	            IF ("gtyp_VGR".horizontal_Axis.di_Actual_Position <= ("gtyp_VGR".di_Pos_MPO_horizontal + "gtyp_VGR".horizontal_Axis.Config.di_Pos_Window))
	                AND ("gtyp_VGR".horizontal_Axis.di_Actual_Position >= ("gtyp_VGR".di_Pos_MPO_horizontal - "gtyp_VGR".horizontal_Axis.Config.di_Pos_Window))
	                AND "gtyp_VGR".horizontal_Axis.x_Position_Reached
	                AND ("gtyp_VGR".vertical_Axis.di_Actual_Position <= ("gtyp_VGR".di_Pos_MPO_vertical - "gtyp_VGR".di_Offset_Pos_MPO_vertical + "gtyp_VGR".vertical_Axis.Config.di_Pos_Window))
	                AND ("gtyp_VGR".vertical_Axis.di_Actual_Position >= ("gtyp_VGR".di_Pos_MPO_vertical - "gtyp_VGR".di_Offset_Pos_MPO_vertical - "gtyp_VGR".vertical_Axis.Config.di_Pos_Window))
	                AND "gtyp_VGR".vertical_Axis.x_Position_Reached THEN
	                "gtyp_VGR".horizontal_Axis.x_Start_Positioning := FALSE;
	                "gtyp_VGR".vertical_Axis.x_Start_Positioning := FALSE;
	                "gtyp_VGR".vertical_Axis.i_PWM := 800;
	                #li_StepCase := 520;
	            END_IF;

	        520: // MPO ready to discard - Position vertical MPO

	            IF "gtyp_MPO".x_Discard_Ready THEN
	                "gtyp_VGR".vertical_Axis.di_Target_Position := "gtyp_VGR".di_Pos_MPO_vertical;
	                "gtyp_VGR".vertical_Axis.x_Start_Positioning := TRUE;
	                "gtyp_VGR".vertical_Axis.i_PWM := 500;

	                IF ("gtyp_VGR".vertical_Axis.di_Actual_Position <= ("gtyp_VGR".di_Pos_MPO_vertical + "gtyp_VGR".vertical_Axis.Config.di_Pos_Window))
	                    AND ("gtyp_VGR".vertical_Axis.di_Actual_Position >= ("gtyp_VGR".di_Pos_MPO_vertical - "gtyp_VGR".vertical_Axis.Config.di_Pos_Window))
	                    AND "gtyp_VGR".vertical_Axis.x_Position_Reached THEN
	                    "gtyp_VGR".vertical_Axis.x_Start_Positioning := FALSE;
	                    "gtyp_VGR".vertical_Axis.i_PWM := 800;
	                    #li_StepCase := 530;
	                    "gtyp_VGR".x_MPO_Req_Discard := FALSE;
	                END_IF;
	            END_IF;

	        530: // turn off vacuum
	            "QX_VGR_ValveVacuum_Q8" := FALSE;
	            #li_StepCase := 540;

	        540: // turn off compressor
	            "QX_VGR_Compressor_Q7" := FALSE;
	            "gtyp_VGR".x_MPO_Discards := TRUE;
	            // Order State
	            "gtyp_VGR".x_Ready_For_Outsource := FALSE;
	            "gtyp_VGR".x_State_Process := TRUE;
	            "gtyp_Interface_Dashboard".Subscribe.State_Order.ldt_ts := DT_TO_LDT(#ldt_MQTT);
	            "gtyp_Interface_Dashboard".Subscribe.State_Order.s_state := 'IN_PROCESS';
	            "gtyp_Interface_Dashboard".Subscribe.State_Order.s_type := "gtyp_VGR".Workpiece.s_type;
	            #li_StepCase := 550;

	        550: // Workpiece discard accepted - Position pre vertical MPO

	            IF "gtyp_MPO".x_MPO_Discards_Accepted THEN
	                "gtyp_VGR".vertical_Axis.di_Target_Position := "gtyp_VGR".di_Pos_MPO_vertical - "gtyp_VGR".di_Offset_Pos_MPO_vertical;
	                "gtyp_VGR".vertical_Axis.x_Start_Positioning := TRUE;
	                "gtyp_VGR".vertical_Axis.i_PWM := 500;

	                IF ("gtyp_VGR".vertical_Axis.di_Actual_Position <= ("gtyp_VGR".di_Pos_MPO_vertical - "gtyp_VGR".di_Offset_Pos_MPO_vertical + "gtyp_VGR".vertical_Axis.Config.di_Pos_Window))
	                    AND ("gtyp_VGR".vertical_Axis.di_Actual_Position >= ("gtyp_VGR".di_Pos_MPO_vertical - "gtyp_VGR".di_Offset_Pos_MPO_vertical - "gtyp_VGR".vertical_Axis.Config.di_Pos_Window))
	                    AND "gtyp_VGR".vertical_Axis.x_Position_Reached THEN
	                    "gtyp_VGR".vertical_Axis.x_Start_Positioning := FALSE;
	                    "gtyp_VGR".x_MPO_Discards := FALSE;
	                    "gtyp_VGR".vertical_Axis.i_PWM := 800;
	                    #li_StepCase := 560;
	                END_IF;
	            END_IF;

	        560: // homing horizontal axis
	            "gtyp_VGR".horizontal_Axis.x_Reference := TRUE;

	            IF NOT "gtyp_VGR".horizontal_Axis.x_Referenced THEN
	                #li_StepCase := 570;
	            END_IF;

	        570: // homed horizontal axis
	            IF "gtyp_VGR".horizontal_Axis.x_Referenced THEN
	                "gtyp_VGR".horizontal_Axis.x_Reference := FALSE;
	                "gtyp_VGR".x_MPO_Discards := FALSE;
	                #li_StepCase := 580;
	            END_IF;

	        580: // wait sequence
	            #lx_Start_TON_Wait := TRUE;
	            #lt_TON_Wait := T#500ms;

	            IF #lfb_TON_Wait.Q THEN
	                "gtyp_VGR".Workpiece.s_id := '0';
	                "gtyp_VGR".Workpiece.s_state := '';
	                "gtyp_VGR".Workpiece.s_type := '';
	                FOR #li_Counter := 1 TO 8 DO
	                    "gtyp_VGR".History[#li_Counter].i_code := 0;
	                    "gtyp_VGR".History[#li_Counter].ldt_ts := DT#1990-01-01-00:00:00;
	                END_FOR;
	                #lx_Start_TON_Wait := FALSE;
	                #li_StepCase := 0;
	            END_IF;

	            (*******************************************************************************************)
	            (**************************      Procedure - store raw parts      **************************)
	            (*******************************************************************************************)

	        600:// approach pick-up position dsi with vertical, horizontal, rotate axis
	            "gtyp_VGR".horizontal_Axis.di_Target_Position := "gtyp_VGR".di_Pos_DSI_horizontal;
	            "gtyp_VGR".horizontal_Axis.x_Start_Positioning := TRUE;
	            "gtyp_VGR".vertical_Axis.di_Target_Position := "gtyp_VGR".di_Pos_DSI_Collect_vertical;
	            "gtyp_VGR".vertical_Axis.x_Start_Positioning := TRUE;
	            "gtyp_VGR".vertical_Axis.i_PWM := 500;
	            "gtyp_VGR".rotate_Axis.di_Target_Position := "gtyp_VGR".di_Pos_DSI_rotate;
	            "gtyp_VGR".rotate_Axis.x_Start_Positioning := TRUE;

	            IF ("gtyp_VGR".horizontal_Axis.di_Actual_Position <= ("gtyp_VGR".di_Pos_DSI_horizontal + "gtyp_VGR".horizontal_Axis.Config.di_Pos_Window))
	                AND ("gtyp_VGR".horizontal_Axis.di_Actual_Position >= ("gtyp_VGR".di_Pos_DSI_horizontal - "gtyp_VGR".horizontal_Axis.Config.di_Pos_Window))
	                AND "gtyp_VGR".horizontal_Axis.x_Position_Reached THEN
	                "gtyp_VGR".horizontal_Axis.x_Start_Positioning := FALSE;
	            END_IF;

	            IF ("gtyp_VGR".vertical_Axis.di_Actual_Position <= ("gtyp_VGR".di_Pos_DSI_Collect_vertical + "gtyp_VGR".vertical_Axis.Config.di_Pos_Window))
	                AND ("gtyp_VGR".vertical_Axis.di_Actual_Position >= ("gtyp_VGR".di_Pos_DSI_Collect_vertical - "gtyp_VGR".vertical_Axis.Config.di_Pos_Window))
	                AND "gtyp_VGR".vertical_Axis.x_Position_Reached THEN
	                "gtyp_VGR".vertical_Axis.x_Start_Positioning := FALSE;
	            END_IF;

	            IF ("gtyp_VGR".rotate_Axis.di_Actual_Position <= ("gtyp_VGR".di_Pos_DSI_rotate + "gtyp_VGR".rotate_Axis.Config.di_Pos_Window))
	                AND ("gtyp_VGR".rotate_Axis.di_Actual_Position >= ("gtyp_VGR".di_Pos_DSI_rotate - "gtyp_VGR".rotate_Axis.Config.di_Pos_Window))
	                AND "gtyp_VGR".rotate_Axis.x_Position_Reached THEN
	                "gtyp_VGR".rotate_Axis.x_Start_Positioning := FALSE;
	            END_IF;

	            IF ("gtyp_VGR".horizontal_Axis.di_Actual_Position <= ("gtyp_VGR".di_Pos_DSI_horizontal + "gtyp_VGR".horizontal_Axis.Config.di_Pos_Window))
	                AND ("gtyp_VGR".horizontal_Axis.di_Actual_Position >= ("gtyp_VGR".di_Pos_DSI_horizontal - "gtyp_VGR".horizontal_Axis.Config.di_Pos_Window))
	                AND "gtyp_VGR".horizontal_Axis.x_Position_Reached
	                AND ("gtyp_VGR".vertical_Axis.di_Actual_Position <= ("gtyp_VGR".di_Pos_DSI_Collect_vertical + "gtyp_VGR".vertical_Axis.Config.di_Pos_Window))
	                AND ("gtyp_VGR".vertical_Axis.di_Actual_Position >= ("gtyp_VGR".di_Pos_DSI_Collect_vertical - "gtyp_VGR".vertical_Axis.Config.di_Pos_Window))
	                AND "gtyp_VGR".vertical_Axis.x_Position_Reached
	                AND ("gtyp_VGR".rotate_Axis.di_Actual_Position <= ("gtyp_VGR".di_Pos_DSI_rotate + "gtyp_VGR".rotate_Axis.Config.di_Pos_Window))
	                AND ("gtyp_VGR".rotate_Axis.di_Actual_Position >= ("gtyp_VGR".di_Pos_DSI_rotate - "gtyp_VGR".rotate_Axis.Config.di_Pos_Window))
	                AND "gtyp_VGR".rotate_Axis.x_Position_Reached THEN
	                "gtyp_VGR".horizontal_Axis.x_Start_Positioning := FALSE;
	                "gtyp_VGR".vertical_Axis.x_Start_Positioning := FALSE;
	                "gtyp_VGR".rotate_Axis.x_Start_Positioning := FALSE;
	                "gtyp_VGR".vertical_Axis.i_PWM := 800;
	                #li_StepCase := 610;
	            END_IF;

	        610:// set status 100 raw goods delivered
	            #li_Return_LDT := RD_SYS_T(#ldt_MQTT);
	            "gtyp_VGR".Workpiece.s_state := 'RAW';
	            "gtyp_VGR".History[1].ldt_ts := DT_TO_LDT(#ldt_MQTT);
	            "gtyp_VGR".History[1].i_code := 100;
	            #li_StepCase := 620;

	        620:// wait sequence
	            #lx_Start_TON_Wait := TRUE;
	            #lt_TON_Wait := T#500ms;

	            IF #lfb_TON_Wait.Q THEN
	                #lx_Start_TON_Wait := FALSE;
	                #li_StepCase := 630;
	            END_IF;

	        630:// turn on compressor and wait
	            "QX_VGR_Compressor_Q7" := TRUE;

	            #lx_Start_TON_Wait := TRUE;
	            #lt_TON_Wait := T#500ms;

	            IF #lfb_TON_Wait.Q THEN
	                #lx_Start_TON_Wait := FALSE;
	                #li_StepCase := 640;
	            END_IF;

	        640:// turn on vacuum
	            "QX_VGR_ValveVacuum_Q8" := true;

	            #li_StepCase := 650;

	        650:// Position vertical NFC
	            #lx_State_activ := TRUE;
	            #ls_Target := 'hbw';

	            "gtyp_VGR".vertical_Axis.di_Target_Position := "gtyp_VGR".di_Pos_NFC_vertical - "gtyp_VGR".di_Offset_Pos_DSI_NFC_vertical;
	            "gtyp_VGR".vertical_Axis.x_Start_Positioning := TRUE;
	            "gtyp_VGR".vertical_Axis.i_PWM := 800;

	            IF ("gtyp_VGR".vertical_Axis.di_Actual_Position <= ("gtyp_VGR".di_Pos_NFC_vertical - "gtyp_VGR".di_Offset_Pos_DSI_NFC_vertical + "gtyp_VGR".vertical_Axis.Config.di_Pos_Window))
	                AND ("gtyp_VGR".vertical_Axis.di_Actual_Position >= ("gtyp_VGR".di_Pos_NFC_vertical - "gtyp_VGR".di_Offset_Pos_DSI_NFC_vertical - "gtyp_VGR".vertical_Axis.Config.di_Pos_Window))
	                AND "gtyp_VGR".vertical_Axis.x_Position_Reached THEN
	                "gtyp_VGR".vertical_Axis.x_Start_Positioning := FALSE;
	                #li_StepCase := 660;
	            END_IF;

	        660: // wait sequence
	            #lx_Start_TON_Wait := TRUE;
	            #lt_TON_Wait := T#500ms;

	            IF #lfb_TON_Wait.Q THEN
	                #lx_Start_TON_Wait := FALSE;
	                #li_StepCase := 670;
	            END_IF;

	        670: // Position horizontal/rotate NFC

	            "gtyp_VGR".horizontal_Axis.di_Target_Position := "gtyp_VGR".di_Pos_NFC_horizontal;
	            "gtyp_VGR".horizontal_Axis.x_Start_Positioning := TRUE;
	            "gtyp_VGR".rotate_Axis.di_Target_Position := "gtyp_VGR".di_Pos_NFC_rotate;
	            "gtyp_VGR".rotate_Axis.x_Start_Positioning := TRUE;

	            IF ("gtyp_VGR".horizontal_Axis.di_Actual_Position <= ("gtyp_VGR".di_Pos_NFC_horizontal + "gtyp_VGR".horizontal_Axis.Config.di_Pos_Window))
	                AND ("gtyp_VGR".horizontal_Axis.di_Actual_Position >= ("gtyp_VGR".di_Pos_NFC_horizontal - "gtyp_VGR".horizontal_Axis.Config.di_Pos_Window))
	                AND "gtyp_VGR".horizontal_Axis.x_Position_Reached THEN
	                "gtyp_VGR".horizontal_Axis.x_Start_Positioning := FALSE;
	            END_IF;

	            IF ("gtyp_VGR".rotate_Axis.di_Actual_Position <= ("gtyp_VGR".di_Pos_NFC_rotate + "gtyp_VGR".rotate_Axis.Config.di_Pos_Window))
	                AND ("gtyp_VGR".rotate_Axis.di_Actual_Position >= ("gtyp_VGR".di_Pos_NFC_rotate - "gtyp_VGR".rotate_Axis.Config.di_Pos_Window))
	                AND "gtyp_VGR".rotate_Axis.x_Position_Reached THEN
	                "gtyp_VGR".rotate_Axis.x_Start_Positioning := FALSE;
	            END_IF;

	            IF ("gtyp_VGR".horizontal_Axis.di_Actual_Position <= ("gtyp_VGR".di_Pos_NFC_horizontal + "gtyp_VGR".horizontal_Axis.Config.di_Pos_Window))
	                AND ("gtyp_VGR".horizontal_Axis.di_Actual_Position >= ("gtyp_VGR".di_Pos_NFC_horizontal - "gtyp_VGR".horizontal_Axis.Config.di_Pos_Window))
	                AND "gtyp_VGR".horizontal_Axis.x_Position_Reached
	                AND ("gtyp_VGR".rotate_Axis.di_Actual_Position <= ("gtyp_VGR".di_Pos_NFC_rotate + "gtyp_VGR".rotate_Axis.Config.di_Pos_Window))
	                AND ("gtyp_VGR".rotate_Axis.di_Actual_Position >= ("gtyp_VGR".di_Pos_NFC_rotate - "gtyp_VGR".rotate_Axis.Config.di_Pos_Window))
	                AND "gtyp_VGR".rotate_Axis.x_Position_Reached THEN
	                "gtyp_VGR".horizontal_Axis.x_Start_Positioning := FALSE;
	                "gtyp_VGR".rotate_Axis.x_Start_Positioning := FALSE;
	                #li_StepCase := 680;
	            END_IF;

	        680: // wait sequence
	            #lx_Start_TON_Wait := TRUE;
	            #lt_TON_Wait := T#500ms;

	            IF #lfb_TON_Wait.Q THEN
	                #lx_Start_TON_Wait := FALSE;
	                #li_StepCase := 690;
	            END_IF;

	        690: // Position vertical NFC

	            "gtyp_VGR".vertical_Axis.di_Target_Position := "gtyp_VGR".di_Pos_NFC_vertical;
	            "gtyp_VGR".vertical_Axis.x_Start_Positioning := TRUE;
	            "gtyp_VGR".vertical_Axis.i_PWM := 500;

	            IF ("gtyp_VGR".vertical_Axis.di_Actual_Position <= ("gtyp_VGR".di_Pos_NFC_vertical + "gtyp_VGR".vertical_Axis.Config.di_Pos_Window))
	                AND ("gtyp_VGR".vertical_Axis.di_Actual_Position >= ("gtyp_VGR".di_Pos_NFC_vertical - "gtyp_VGR".vertical_Axis.Config.di_Pos_Window))
	                AND "gtyp_VGR".vertical_Axis.x_Position_Reached THEN
	                "gtyp_VGR".vertical_Axis.x_Start_Positioning := FALSE;
	                "gtyp_VGR".vertical_Axis.i_PWM := 800;
	                #li_StepCase := 700;
	            END_IF;

	        700: // Start delete/write/read NFC
	            "gtyp_VGR".x_NFC_Start_First := TRUE;

	            IF "gtyp_VGR".x_NFC_Completed THEN
	                "gtyp_VGR".x_NFC_Start_First := FALSE;
	                #li_StepCase := 710;
	            END_IF;

	        710: // Position vertical pre NFC

	            "gtyp_VGR".vertical_Axis.di_Target_Position := "gtyp_VGR".di_Pos_NFC_vertical - "gtyp_VGR".di_Offset_Pos_DSI_NFC_vertical;
	            "gtyp_VGR".vertical_Axis.x_Start_Positioning := TRUE;
	            "gtyp_VGR".vertical_Axis.i_PWM := 800;

	            IF ("gtyp_VGR".vertical_Axis.di_Actual_Position <= ("gtyp_VGR".di_Pos_NFC_vertical - "gtyp_VGR".di_Offset_Pos_DSI_NFC_vertical + "gtyp_VGR".vertical_Axis.Config.di_Pos_Window))
	                AND ("gtyp_VGR".vertical_Axis.di_Actual_Position >= ("gtyp_VGR".di_Pos_NFC_vertical - "gtyp_VGR".di_Offset_Pos_DSI_NFC_vertical - "gtyp_VGR".vertical_Axis.Config.di_Pos_Window))
	                AND "gtyp_VGR".vertical_Axis.x_Position_Reached THEN
	                "gtyp_VGR".vertical_Axis.x_Start_Positioning := FALSE;
	                #li_StepCase := 720;
	            END_IF;

	        720: // Position horizontal/rotate Color

	            "gtyp_VGR".horizontal_Axis.di_Target_Position := "gtyp_VGR".di_Pos_Color_horizontal;
	            "gtyp_VGR".horizontal_Axis.x_Start_Positioning := TRUE;
	            "gtyp_VGR".rotate_Axis.di_Target_Position := "gtyp_VGR".di_Pos_Color_rotate;
	            "gtyp_VGR".rotate_Axis.x_Start_Positioning := TRUE;

	            IF ("gtyp_VGR".horizontal_Axis.di_Actual_Position <= ("gtyp_VGR".di_Pos_Color_horizontal + "gtyp_VGR".horizontal_Axis.Config.di_Pos_Window))
	                AND ("gtyp_VGR".horizontal_Axis.di_Actual_Position >= ("gtyp_VGR".di_Pos_Color_horizontal - "gtyp_VGR".horizontal_Axis.Config.di_Pos_Window))
	                AND "gtyp_VGR".horizontal_Axis.x_Position_Reached THEN
	                "gtyp_VGR".horizontal_Axis.x_Start_Positioning := FALSE;
	            END_IF;

	            IF ("gtyp_VGR".rotate_Axis.di_Actual_Position <= ("gtyp_VGR".di_Pos_Color_rotate + "gtyp_VGR".rotate_Axis.Config.di_Pos_Window))
	                AND ("gtyp_VGR".rotate_Axis.di_Actual_Position >= ("gtyp_VGR".di_Pos_Color_rotate - "gtyp_VGR".rotate_Axis.Config.di_Pos_Window))
	                AND "gtyp_VGR".rotate_Axis.x_Position_Reached THEN
	                "gtyp_VGR".rotate_Axis.x_Start_Positioning := FALSE;
	            END_IF;

	            IF ("gtyp_VGR".horizontal_Axis.di_Actual_Position <= ("gtyp_VGR".di_Pos_Color_horizontal + "gtyp_VGR".horizontal_Axis.Config.di_Pos_Window))
	                AND ("gtyp_VGR".horizontal_Axis.di_Actual_Position >= ("gtyp_VGR".di_Pos_Color_horizontal - "gtyp_VGR".horizontal_Axis.Config.di_Pos_Window))
	                AND "gtyp_VGR".horizontal_Axis.x_Position_Reached
	                AND ("gtyp_VGR".rotate_Axis.di_Actual_Position <= ("gtyp_VGR".di_Pos_Color_rotate + "gtyp_VGR".rotate_Axis.Config.di_Pos_Window))
	                AND ("gtyp_VGR".rotate_Axis.di_Actual_Position >= ("gtyp_VGR".di_Pos_Color_rotate - "gtyp_VGR".rotate_Axis.Config.di_Pos_Window))
	                AND "gtyp_VGR".rotate_Axis.x_Position_Reached THEN
	                "gtyp_VGR".horizontal_Axis.x_Start_Positioning := FALSE;
	                "gtyp_VGR".rotate_Axis.x_Start_Positioning := FALSE;
	                #li_StepCase := 730;
	            END_IF;

	        730: // wait sequence
	            #lx_Start_TON_Wait := TRUE;
	            #lt_TON_Wait := T#500ms;

	            IF #lfb_TON_Wait.Q THEN
	                #lx_Start_TON_Wait := FALSE;
	                #li_StepCase := 740;
	            END_IF;

	        740: // Position vertical Color
	            "gtyp_VGR".vertical_Axis.di_Target_Position := "gtyp_VGR".di_Pos_Color_vertical;
	            "gtyp_VGR".vertical_Axis.x_Start_Positioning := TRUE;
	            "gtyp_VGR".vertical_Axis.i_PWM := 500;

	            IF ("gtyp_VGR".vertical_Axis.di_Actual_Position <= ("gtyp_VGR".di_Pos_Color_vertical + "gtyp_VGR".vertical_Axis.Config.di_Pos_Window))
	                AND ("gtyp_VGR".vertical_Axis.di_Actual_Position >= ("gtyp_VGR".di_Pos_Color_vertical - "gtyp_VGR".vertical_Axis.Config.di_Pos_Window))
	                AND "gtyp_VGR".vertical_Axis.x_Position_Reached THEN
	                "gtyp_VGR".vertical_Axis.x_Start_Positioning := FALSE;
	                "gtyp_VGR".vertical_Axis.i_PWM := 800;
	                #li_StepCase := 750;
	            END_IF;

	        750: // evaluate color workpiece
	            #ls_Color := '';

	            IF "IW_SSC_ColorSensor_A1" >= "gtyp_SSC".w_Threshold_Red_Blue THEN
	                //               IF "IW_SSC_ColorSensor" > 16000 AND "IW_SSC_ColorSensor" < 17500 THEN
	                #ls_Color := 'BLUE';
	            ELSIF "IW_SSC_ColorSensor_A1" <= "gtyp_SSC".w_Threshold_White_Red THEN
	                //            ELSIF "IW_SSC_ColorSensor" > 5000 AND "IW_SSC_ColorSensor" < 11000 THEN
	                #ls_Color := 'WHITE';
	            ELSIF "IW_SSC_ColorSensor_A1" > "gtyp_SSC".w_Threshold_White_Red AND "IW_SSC_ColorSensor_A1" < "gtyp_SSC".w_Threshold_Red_Blue THEN
	                //            ELSIF "IW_SSC_ColorSensor" > 11000 AND "IW_SSC_ColorSensor" < 16000 THEN
	                #ls_Color := 'RED';
	            END_IF;

	            #li_Return_LDT := RD_SYS_T(#ldt_MQTT);
	            "gtyp_VGR".History[2].ldt_ts := DT_TO_LDT(#ldt_MQTT);
	            "gtyp_VGR".History[2].i_code := 200;
	            "gtyp_VGR".Workpiece.s_type := #ls_Color;

	            #lx_Start_TON_Wait := TRUE;
	            #lt_TON_Wait := T#500ms;

	            IF #lfb_TON_Wait.Q THEN
	                #lx_Start_TON_Wait := FALSE;
	                #li_StepCase := 760;
	            END_IF;

	        760: // Position vertical pre NFC
	            "gtyp_VGR".vertical_Axis.di_Target_Position := "gtyp_VGR".di_Pos_NFC_vertical - "gtyp_VGR".di_Offset_Pos_DSI_NFC_vertical;
	            "gtyp_VGR".vertical_Axis.x_Start_Positioning := TRUE;
	            "gtyp_VGR".vertical_Axis.i_PWM := 500;

	            IF ("gtyp_VGR".vertical_Axis.di_Actual_Position <= ("gtyp_VGR".di_Pos_NFC_vertical - "gtyp_VGR".di_Offset_Pos_DSI_NFC_vertical + "gtyp_VGR".vertical_Axis.Config.di_Pos_Window))
	                AND ("gtyp_VGR".vertical_Axis.di_Actual_Position >= ("gtyp_VGR".di_Pos_NFC_vertical - "gtyp_VGR".di_Offset_Pos_DSI_NFC_vertical - "gtyp_VGR".vertical_Axis.Config.di_Pos_Window))
	                AND "gtyp_VGR".vertical_Axis.x_Position_Reached THEN
	                "gtyp_VGR".vertical_Axis.x_Start_Positioning := FALSE;
	                "gtyp_VGR".vertical_Axis.i_PWM := 800;
	                #li_StepCase := 770;
	            END_IF;

	        770: // wait sequence
	            #lx_Start_TON_Wait := TRUE;
	            #lt_TON_Wait := T#500ms;

	            IF #lfb_TON_Wait.Q THEN
	                #lx_Start_TON_Wait := FALSE;
	                #li_StepCase := 780;
	            END_IF;

	        780: // Position horizontal/rotate NFC

	            "gtyp_VGR".horizontal_Axis.di_Target_Position := "gtyp_VGR".di_Pos_NFC_horizontal;
	            "gtyp_VGR".horizontal_Axis.x_Start_Positioning := TRUE;
	            "gtyp_VGR".rotate_Axis.di_Target_Position := "gtyp_VGR".di_Pos_NFC_rotate;
	            "gtyp_VGR".rotate_Axis.x_Start_Positioning := TRUE;

	            IF ("gtyp_VGR".horizontal_Axis.di_Actual_Position <= ("gtyp_VGR".di_Pos_NFC_horizontal + "gtyp_VGR".horizontal_Axis.Config.di_Pos_Window))
	                AND ("gtyp_VGR".horizontal_Axis.di_Actual_Position >= ("gtyp_VGR".di_Pos_NFC_horizontal - "gtyp_VGR".horizontal_Axis.Config.di_Pos_Window))
	                AND "gtyp_VGR".horizontal_Axis.x_Position_Reached THEN
	                "gtyp_VGR".horizontal_Axis.x_Start_Positioning := FALSE;
	            END_IF;

	            IF ("gtyp_VGR".rotate_Axis.di_Actual_Position <= ("gtyp_VGR".di_Pos_NFC_rotate + "gtyp_VGR".rotate_Axis.Config.di_Pos_Window))
	                AND ("gtyp_VGR".rotate_Axis.di_Actual_Position >= ("gtyp_VGR".di_Pos_NFC_rotate - "gtyp_VGR".rotate_Axis.Config.di_Pos_Window))
	                AND "gtyp_VGR".rotate_Axis.x_Position_Reached THEN
	                "gtyp_VGR".rotate_Axis.x_Start_Positioning := FALSE;
	            END_IF;

	            IF ("gtyp_VGR".horizontal_Axis.di_Actual_Position <= ("gtyp_VGR".di_Pos_NFC_horizontal + "gtyp_VGR".horizontal_Axis.Config.di_Pos_Window))
	                AND ("gtyp_VGR".horizontal_Axis.di_Actual_Position >= ("gtyp_VGR".di_Pos_NFC_horizontal - "gtyp_VGR".horizontal_Axis.Config.di_Pos_Window))
	                AND "gtyp_VGR".horizontal_Axis.x_Position_Reached
	                AND ("gtyp_VGR".rotate_Axis.di_Actual_Position <= ("gtyp_VGR".di_Pos_NFC_rotate + "gtyp_VGR".rotate_Axis.Config.di_Pos_Window))
	                AND ("gtyp_VGR".rotate_Axis.di_Actual_Position >= ("gtyp_VGR".di_Pos_NFC_rotate - "gtyp_VGR".rotate_Axis.Config.di_Pos_Window))
	                AND "gtyp_VGR".rotate_Axis.x_Position_Reached THEN
	                "gtyp_VGR".horizontal_Axis.x_Start_Positioning := FALSE;
	                "gtyp_VGR".vertical_Axis.x_Start_Positioning := FALSE;
	                "gtyp_VGR".rotate_Axis.x_Start_Positioning := FALSE;
	                #li_StepCase := 790;
	            END_IF;

	        790: // wait sequence
	            #lx_Start_TON_Wait := TRUE;
	            #lt_TON_Wait := T#500ms;

	            IF #lfb_TON_Wait.Q THEN
	                #lx_Start_TON_Wait := FALSE;
	                #li_StepCase := 800;
	            END_IF;

	        800: // Position vertical NFC

	            "gtyp_VGR".vertical_Axis.di_Target_Position := "gtyp_VGR".di_Pos_NFC_vertical;
	            "gtyp_VGR".vertical_Axis.x_Start_Positioning := TRUE;
	            "gtyp_VGR".vertical_Axis.i_PWM := 500;

	            IF ("gtyp_VGR".vertical_Axis.di_Actual_Position <= ("gtyp_VGR".di_Pos_NFC_vertical + "gtyp_VGR".vertical_Axis.Config.di_Pos_Window))
	                AND ("gtyp_VGR".vertical_Axis.di_Actual_Position >= ("gtyp_VGR".di_Pos_NFC_vertical - "gtyp_VGR".vertical_Axis.Config.di_Pos_Window))
	                AND "gtyp_VGR".vertical_Axis.x_Position_Reached THEN
	                "gtyp_VGR".vertical_Axis.x_Start_Positioning := FALSE;
	                "gtyp_VGR".vertical_Axis.i_PWM := 800;
	                #li_StepCase := 810;
	            END_IF;

	        810: // Start write/read NFC Color

	            "gtyp_VGR".x_NFC_Start := TRUE;

	            IF "gtyp_VGR".x_NFC_Completed THEN
	                "gtyp_VGR".x_NFC_Start := FALSE;
	                #li_StepCase := 820;
	            END_IF;

	        820: // Position vertical pre NFC

	            "gtyp_VGR".vertical_Axis.di_Target_Position := "gtyp_VGR".di_Pos_NFC_vertical - "gtyp_VGR".di_Offset_Pos_DSI_NFC_vertical;
	            "gtyp_VGR".vertical_Axis.x_Start_Positioning := TRUE;
	            "gtyp_VGR".vertical_Axis.i_PWM := 500;

	            IF ("gtyp_VGR".vertical_Axis.di_Actual_Position <= ("gtyp_VGR".di_Pos_NFC_vertical - "gtyp_VGR".di_Offset_Pos_DSI_NFC_vertical + "gtyp_VGR".vertical_Axis.Config.di_Pos_Window))
	                AND ("gtyp_VGR".vertical_Axis.di_Actual_Position >= ("gtyp_VGR".di_Pos_NFC_vertical - "gtyp_VGR".di_Offset_Pos_DSI_NFC_vertical - "gtyp_VGR".vertical_Axis.Config.di_Pos_Window))
	                AND "gtyp_VGR".vertical_Axis.x_Position_Reached THEN
	                "gtyp_VGR".vertical_Axis.x_Start_Positioning := FALSE;
	                "gtyp_VGR".vertical_Axis.i_PWM := 800;
	                #li_StepCase := 830;
	            END_IF;

	        830: // wait sequence
	            #lx_Start_TON_Wait := TRUE;
	            #lt_TON_Wait := T#500ms;

	            IF #lfb_TON_Wait.Q THEN
	                #lx_Start_TON_Wait := FALSE;
	                #li_StepCase := 840;
	            END_IF;

	        840: // Position rotate HBW and homing horizontal/vertical axis
	            "gtyp_VGR".rotate_Axis.di_Target_Position := "gtyp_VGR".di_Pos_HBW_rotate;
	            "gtyp_VGR".rotate_Axis.x_Start_Positioning := TRUE;

	            "gtyp_VGR".horizontal_Axis.x_Reference := TRUE;
	            "gtyp_VGR".vertical_Axis.x_Reference := TRUE;

	            IF ("gtyp_VGR".rotate_Axis.di_Actual_Position <= ("gtyp_VGR".di_Pos_HBW_rotate + "gtyp_VGR".rotate_Axis.Config.di_Pos_Window))
	                AND ("gtyp_VGR".rotate_Axis.di_Actual_Position >= ("gtyp_VGR".di_Pos_HBW_rotate - "gtyp_VGR".rotate_Axis.Config.di_Pos_Window))
	                AND "gtyp_VGR".rotate_Axis.x_Position_Reached THEN
	                "gtyp_VGR".rotate_Axis.x_Start_Positioning := FALSE;
	            END_IF;

	            IF NOT "gtyp_VGR".horizontal_Axis.x_Referenced AND NOT "gtyp_VGR".vertical_Axis.x_Referenced THEN
	                #li_StepCase := 850;
	            END_IF;

	        850: // Position rotate HBW reached and homed horizontal/vertical axis

	            IF ("gtyp_VGR".rotate_Axis.di_Actual_Position <= ("gtyp_VGR".di_Pos_HBW_rotate + "gtyp_VGR".rotate_Axis.Config.di_Pos_Window))
	                AND ("gtyp_VGR".rotate_Axis.di_Actual_Position >= ("gtyp_VGR".di_Pos_HBW_rotate - "gtyp_VGR".rotate_Axis.Config.di_Pos_Window))
	                AND "gtyp_VGR".rotate_Axis.x_Position_Reached THEN
	                "gtyp_VGR".rotate_Axis.x_Start_Positioning := FALSE;
	            END_IF;

	            IF "gtyp_VGR".horizontal_Axis.x_Referenced THEN
	                "gtyp_VGR".horizontal_Axis.x_Reference := FALSE;
	            END_IF;
	            IF "gtyp_VGR".vertical_Axis.x_Referenced THEN
	                "gtyp_VGR".vertical_Axis.x_Reference := FALSE;
	            END_IF;
	            IF "gtyp_VGR".horizontal_Axis.x_Referenced
	                AND "gtyp_VGR".vertical_Axis.x_Referenced
	                AND ("gtyp_VGR".rotate_Axis.di_Actual_Position <= ("gtyp_VGR".di_Pos_HBW_rotate + "gtyp_VGR".rotate_Axis.Config.di_Pos_Window))
	                AND ("gtyp_VGR".rotate_Axis.di_Actual_Position >= ("gtyp_VGR".di_Pos_HBW_rotate - "gtyp_VGR".rotate_Axis.Config.di_Pos_Window))
	                AND "gtyp_VGR".rotate_Axis.x_Position_Reached THEN
	                "gtyp_VGR".horizontal_Axis.x_Reference := FALSE;
	                "gtyp_VGR".vertical_Axis.x_Reference := FALSE;
	                "gtyp_VGR".rotate_Axis.x_Start_Positioning := FALSE;
	                #li_StepCase := 860;
	            END_IF;

	        860: // wait sequence
	            #lx_Start_TON_Wait := TRUE;
	            #lt_TON_Wait := T#500ms;

	            IF #lfb_TON_Wait.Q THEN
	                #lx_Start_TON_Wait := FALSE;
	                #li_StepCase := 870;
	            END_IF;

	        870: // Position horizontal HBW

	            "gtyp_VGR".horizontal_Axis.di_Target_Position := "gtyp_VGR".di_Pos_HBW_horizontal;
	            "gtyp_VGR".horizontal_Axis.x_Start_Positioning := TRUE;

	            IF ("gtyp_VGR".horizontal_Axis.di_Actual_Position <= ("gtyp_VGR".di_Pos_HBW_horizontal + "gtyp_VGR".horizontal_Axis.Config.di_Pos_Window))
	                AND ("gtyp_VGR".horizontal_Axis.di_Actual_Position >= ("gtyp_VGR".di_Pos_HBW_horizontal - "gtyp_VGR".horizontal_Axis.Config.di_Pos_Window))
	                AND "gtyp_VGR".horizontal_Axis.x_Position_Reached THEN
	                "gtyp_VGR".horizontal_Axis.x_Start_Positioning := FALSE;
	                #li_StepCase := 880;
	            END_IF;

	        880: // container available start drop down
	            IF "gtyp_HBW".x_HBW_Container_Available THEN
	                #li_StepCase := 890;
	            END_IF;

	        890: // Position vertical discard HBW
	            "gtyp_VGR".vertical_Axis.di_Target_Position := "gtyp_VGR".di_Pos_HBW_Discard_vertical;
	            "gtyp_VGR".vertical_Axis.x_Start_Positioning := TRUE;
	            "gtyp_VGR".vertical_Axis.i_PWM := 500;

	            IF ("gtyp_VGR".vertical_Axis.di_Actual_Position <= ("gtyp_VGR".di_Pos_HBW_Discard_vertical + "gtyp_VGR".vertical_Axis.Config.di_Pos_Window))
	                AND ("gtyp_VGR".vertical_Axis.di_Actual_Position >= ("gtyp_VGR".di_Pos_HBW_Discard_vertical - "gtyp_VGR".vertical_Axis.Config.di_Pos_Window))
	                AND "gtyp_VGR".vertical_Axis.x_Position_Reached THEN
	                "gtyp_VGR".vertical_Axis.x_Start_Positioning := FALSE;
	                "gtyp_VGR".vertical_Axis.i_PWM := 800;
	                #li_StepCase := 900;
	            END_IF;

	        900: // turn off vacuum
	            "QX_VGR_ValveVacuum_Q8" := FALSE;
	            #li_StepCase := 910;

	        910: // turn off compressor
	            "QX_VGR_Compressor_Q7" := FALSE;
	            "gtyp_VGR".x_HBW_Discards := TRUE;

	            #lx_Start_TON_Wait := TRUE;
	            #lt_TON_Wait := T#500ms;

	            IF #lfb_TON_Wait.Q AND "gtyp_HBW".x_HBW_Discards_Accepted THEN
	                #lx_State_activ := FALSE;
	                #ls_Target := '';
	                "gtyp_VGR".x_HBW_Discards := FALSE;
	                "gtyp_VGR".x_HBW_Storage := FALSE;
	                #lx_Start_TON_Wait := FALSE;
	                #li_StepCase := 920;
	            END_IF;

	        920: // homing vertical axis
	            "gtyp_VGR".vertical_Axis.x_Reference := TRUE;

	            IF NOT "gtyp_VGR".vertical_Axis.x_Referenced THEN
	                #li_StepCase := 930;
	            END_IF;

	        930: // homed vertical axis
	            IF "gtyp_VGR".vertical_Axis.x_Referenced THEN
	                "gtyp_VGR".vertical_Axis.x_Reference := FALSE;
	                #li_StepCase := 940;
	            END_IF;

	        940: // homing horizontal axis
	            "gtyp_VGR".horizontal_Axis.x_Reference := TRUE;

	            IF NOT "gtyp_VGR".horizontal_Axis.x_Referenced THEN
	                #li_StepCase := 950;
	            END_IF;

	        950: // homed horizontal axis
	            IF "gtyp_VGR".horizontal_Axis.x_Referenced THEN
	                "gtyp_VGR".horizontal_Axis.x_Reference := FALSE;
	                #li_StepCase := 960;
	            END_IF;

	        960: // wait sequence
	            #lx_Start_TON_Wait := TRUE;
	            #lt_TON_Wait := T#500ms;

	            IF #lfb_TON_Wait.Q AND "gtyp_HBW".x_HBW_Discards_Accepted THEN
	                "gtyp_VGR".x_HBW_Discards := FALSE;
	                #lx_Start_TON_Wait := FALSE;
	                "gtyp_VGR".Workpiece.s_id := '';
	                "gtyp_VGR".Workpiece.s_state := '';
	                "gtyp_VGR".Workpiece.s_type := '';
	                FOR #li_Counter := 1 TO 8 DO
	                    // Statement section FOR
	                    "gtyp_VGR".History[#li_Counter].i_code := 0;
	                    "gtyp_VGR".History[#li_Counter].ldt_ts := DT#1990-01-01-00:00:00;
	                END_FOR;
	                #li_StepCase := 0;
	            END_IF;

	        1200:// homing vertical axis
	            "gtyp_VGR".Workpiece.s_id := '0';
	            "gtyp_VGR".Workpiece.s_state := '';
	            "gtyp_VGR".Workpiece.s_type := '';
	            FOR #li_Counter := 1 TO 8 DO
	                "gtyp_VGR".History[#li_Counter].i_code := 0;
	                "gtyp_VGR".History[#li_Counter].ldt_ts := DT#1990-01-01-00:00:00;
	            END_FOR;

	            IF "gtyp_HBW".x_HBW_Container_Available THEN
	                "gtyp_VGR".x_HBW_Discards := TRUE;
	            END_IF;

	            IF "gtyp_HBW".x_HBW_Discards_Accepted OR "gtyp_HBW".x_HBW_PickedUp_Accepted THEN
	                "gtyp_VGR".x_HBW_Discards := FALSE;
	                "gtyp_VGR".x_HBW_PickedUp := FALSE;
	                "gtyp_HBW".x_HBW_Discards_Accepted := FALSE;
	                "gtyp_HBW".x_HBW_PickedUp_Accepted := FALSE;
	            END_IF;

	            #li_Lights := 2;
	            "gtyp_VGR".vertical_Axis.x_Reference := TRUE;

	            IF NOT "gtyp_VGR".vertical_Axis.x_Referenced THEN
	                #li_StepCase := 1210;
	            END_IF;

	        1210: // homed vertical axis
	            IF "gtyp_VGR".vertical_Axis.x_Referenced THEN
	                "gtyp_VGR".vertical_Axis.x_Reference := FALSE;
	                #li_StepCase := 1220;
	            END_IF;

	        1220: // homing horizontal axis
	            "gtyp_VGR".horizontal_Axis.x_Reference := TRUE;

	            IF NOT "gtyp_VGR".horizontal_Axis.x_Referenced THEN
	                #li_StepCase := 1230;
	            END_IF;

	        1230: // homed horizontal axis
	            IF "gtyp_VGR".horizontal_Axis.x_Referenced THEN
	                "gtyp_VGR".horizontal_Axis.x_Reference := FALSE;
	                #li_StepCase := 1240;
	            END_IF;

	        1240: // homing rotate axis
	            "gtyp_VGR".rotate_Axis.x_Reference := TRUE;

	            IF NOT "gtyp_VGR".rotate_Axis.x_Referenced THEN
	                #li_StepCase := 1250;
	            END_IF;

	        1250: // homed horizontal axis
	            IF "gtyp_VGR".rotate_Axis.x_Referenced THEN
	                "gtyp_VGR".rotate_Axis.x_Reference := FALSE;
	                #li_StepCase := 1260;
	            END_IF;

	        1260: // Position vertical/horizontal/rotate NiO
	            "gtyp_VGR".horizontal_Axis.di_Target_Position := "gtyp_VGR".di_Pos_NiO_horizontal;
	            "gtyp_VGR".horizontal_Axis.x_Start_Positioning := TRUE;
	            "gtyp_VGR".vertical_Axis.di_Target_Position := "gtyp_VGR".di_Pos_NiO_vertical;
	            "gtyp_VGR".vertical_Axis.x_Start_Positioning := TRUE;
	            "gtyp_VGR".vertical_Axis.i_PWM := 500;
	            "gtyp_VGR".rotate_Axis.di_Target_Position := "gtyp_VGR".di_Pos_NiO_rotate;
	            "gtyp_VGR".rotate_Axis.x_Start_Positioning := TRUE;

	            IF ("gtyp_VGR".horizontal_Axis.di_Actual_Position <= ("gtyp_VGR".di_Pos_NiO_horizontal + "gtyp_VGR".horizontal_Axis.Config.di_Pos_Window))
	                AND ("gtyp_VGR".horizontal_Axis.di_Actual_Position >= ("gtyp_VGR".di_Pos_NiO_horizontal - "gtyp_VGR".horizontal_Axis.Config.di_Pos_Window))
	                AND "gtyp_VGR".horizontal_Axis.x_Position_Reached THEN
	                "gtyp_VGR".horizontal_Axis.x_Start_Positioning := FALSE;
	            END_IF;

	            IF ("gtyp_VGR".vertical_Axis.di_Actual_Position <= ("gtyp_VGR".di_Pos_NiO_vertical + "gtyp_VGR".vertical_Axis.Config.di_Pos_Window))
	                AND ("gtyp_VGR".vertical_Axis.di_Actual_Position >= ("gtyp_VGR".di_Pos_NiO_vertical - "gtyp_VGR".vertical_Axis.Config.di_Pos_Window))
	                AND "gtyp_VGR".vertical_Axis.x_Position_Reached THEN
	                "gtyp_VGR".vertical_Axis.x_Start_Positioning := FALSE;
	            END_IF;

	            IF ("gtyp_VGR".rotate_Axis.di_Actual_Position <= ("gtyp_VGR".di_Pos_NiO_rotate + "gtyp_VGR".rotate_Axis.Config.di_Pos_Window))
	                AND ("gtyp_VGR".rotate_Axis.di_Actual_Position >= ("gtyp_VGR".di_Pos_NiO_rotate - "gtyp_VGR".rotate_Axis.Config.di_Pos_Window))
	                AND "gtyp_VGR".rotate_Axis.x_Position_Reached THEN
	                "gtyp_VGR".rotate_Axis.x_Start_Positioning := FALSE;
	            END_IF;

	            IF ("gtyp_VGR".horizontal_Axis.di_Actual_Position <= ("gtyp_VGR".di_Pos_NiO_horizontal + "gtyp_VGR".horizontal_Axis.Config.di_Pos_Window))
	                AND ("gtyp_VGR".horizontal_Axis.di_Actual_Position >= ("gtyp_VGR".di_Pos_NiO_horizontal - "gtyp_VGR".horizontal_Axis.Config.di_Pos_Window))
	                AND "gtyp_VGR".horizontal_Axis.x_Position_Reached
	                AND ("gtyp_VGR".vertical_Axis.di_Actual_Position <= ("gtyp_VGR".di_Pos_NiO_vertical + "gtyp_VGR".vertical_Axis.Config.di_Pos_Window))
	                AND ("gtyp_VGR".vertical_Axis.di_Actual_Position >= ("gtyp_VGR".di_Pos_NiO_vertical - "gtyp_VGR".vertical_Axis.Config.di_Pos_Window))
	                AND "gtyp_VGR".vertical_Axis.x_Position_Reached
	                AND ("gtyp_VGR".rotate_Axis.di_Actual_Position <= ("gtyp_VGR".di_Pos_NiO_rotate + "gtyp_VGR".rotate_Axis.Config.di_Pos_Window))
	                AND ("gtyp_VGR".rotate_Axis.di_Actual_Position >= ("gtyp_VGR".di_Pos_NiO_rotate - "gtyp_VGR".rotate_Axis.Config.di_Pos_Window))
	                AND "gtyp_VGR".rotate_Axis.x_Position_Reached THEN
	                "gtyp_VGR".horizontal_Axis.x_Start_Positioning := FALSE;
	                "gtyp_VGR".vertical_Axis.x_Start_Positioning := FALSE;
	                "gtyp_VGR".rotate_Axis.x_Start_Positioning := FALSE;
	                "gtyp_VGR".vertical_Axis.i_PWM := 800;
	                #li_StepCase := 1270;
	            END_IF;

	        1270: // turn off vacuum
	            "QX_VGR_ValveVacuum_Q8" := FALSE;
	            #li_StepCase := 1280;

	        1280: // turn off compressor

	            #lx_Start_TON_Wait := TRUE;
	            #lt_TON_Wait := T#1000ms;

	            IF #lfb_TON_Wait.Q THEN
	                "QX_VGR_Compressor_Q7" := FALSE;
	                #lx_Start_TON_Wait := FALSE;
	                "gtyp_VGR".x_Workpiece_NiO := FALSE;
	                "gtyp_VGR".x_HBW_Discards := FALSE;
	                #li_Lights := 1;
	                #li_StepCase := 0;
	            END_IF;
	            // Statement section ELSE
	        ELSE
	            ;
	    END_CASE;

	ELSE
	    "gtyp_VGR".Workpiece.s_id := '';
	    "gtyp_VGR".Workpiece.s_state := '';
	    "gtyp_VGR".Workpiece.s_type := '';
	    // Order State
	    "gtyp_VGR".x_State_Process := FALSE;
	    "gtyp_Interface_Dashboard".Subscribe.State_Order.ldt_ts := DT_TO_LDT(#ldt_MQTT);
	    "gtyp_Interface_Dashboard".Subscribe.State_Order.s_state := 'WAITING_FOR_ORDER';
	    "gtyp_Interface_Dashboard".Subscribe.State_Order.s_type := '';
	    FOR #li_Counter := 1 TO 8 DO
	        "gtyp_VGR".History[#li_Counter].i_code := 0;
	        "gtyp_VGR".History[#li_Counter].ldt_ts := DT#1990-01-01-00:00:00;
	    END_FOR;

	    "gtyp_VGR".x_Start_Park_Position := FALSE;
	    "gtyp_VGR".x_Park_Position_Reached := FALSE;
	    "gtyp_VGR".x_NFC_Start_First := FALSE;
	    "gtyp_VGR".x_NFC_Start := FALSE;
	    "gtyp_VGR".x_NFC_Completed := FALSE;
	    "gtyp_VGR".x_HBW_Storage := FALSE;
	    "gtyp_VGR".x_HBW_Outsource := FALSE;
	    "gtyp_VGR".s_HBW_Outsource_Typ := '';
	    "gtyp_VGR".x_HBW_Discards := FALSE;
	    "gtyp_VGR".x_HBW_PickedUp := FALSE;
	    "gtyp_VGR".x_MPO_Req_Discard := FALSE;
	    "gtyp_VGR".x_MPO_Discards := FALSE;
	    "gtyp_VGR".x_Ready_For_Outsource := FALSE;
	    "gtyp_VGR".x_State_Process := FALSE;
	    "gtyp_VGR".x_Workpiece_NiO := FALSE;

	    "gtyp_VGR".vertical_Axis.i_PWM := 800;

	    #li_Lights := 1;
	    #lx_Init := TRUE;
	END_IF;
END_FUNCTION_BLOCK

FUNCTION_BLOCK "PRG_SSC_Light"
TITLE = Program Lights
{ S7_Optimized_Access := 'TRUE' }
AUTHOR : 'A.Schaefer'
VERSION : 0.0
   VAR
      lx_Init { ExternalAccessible := 'False'; ExternalVisible := 'False'; ExternalWritable := 'False'} : Bool;
      lx_Start { ExternalAccessible := 'False'; ExternalVisible := 'False'; ExternalWritable := 'False'} : Bool;
      li_StepCase { ExternalAccessible := 'False'; ExternalVisible := 'False'; ExternalWritable := 'False'} : Int;
      ldt_MQTT { ExternalAccessible := 'False'; ExternalVisible := 'False'; ExternalWritable := 'False'} : Date_And_Time;
      lldt_ts_old { ExternalAccessible := 'False'; ExternalVisible := 'False'; ExternalWritable := 'False'} : LDT;
      li_Return_LDT { ExternalAccessible := 'False'; ExternalVisible := 'False'; ExternalWritable := 'False'} : Int;
      lfb_TOF_Camera {InstructionName := 'TOF_TIME'; LibVersion := '1.0'; ExternalAccessible := 'False'; ExternalVisible := 'False'; ExternalWritable := 'False'; S7_SetPoint := 'False'} : TOF_TIME;
      lfb_TON_Schritt {InstructionName := 'TON_TIME'; LibVersion := '1.0'; ExternalAccessible := 'False'; ExternalVisible := 'False'; ExternalWritable := 'False'; S7_SetPoint := 'False'} : TON_TIME;
      lfb_blinker_cam { ExternalAccessible := 'False'; ExternalVisible := 'False'; ExternalWritable := 'False'; S7_SetPoint := 'False'} : "FB_Blinker";
      lfb_blinker_config { ExternalAccessible := 'False'; ExternalVisible := 'False'; ExternalWritable := 'False'; S7_SetPoint := 'False'} : "FB_Blinker";
      lx_StartTimer { ExternalAccessible := 'False'; ExternalVisible := 'False'; ExternalWritable := 'False'} : Bool;
   END_VAR


BEGIN
	IF #lx_Init THEN

	    // if camera sen picture - Red light flash
	    IF "gtyp_Interface_Dashboard".Subscribe.CameraPicture.ldt_ts > #lldt_ts_old THEN
	        #lldt_ts_old := "gtyp_Interface_Dashboard".Subscribe.CameraPicture.ldt_ts;
	        #lfb_blinker_cam(int_periodendauer := T#50ms);
	    END_IF;

	    // reload flash
	    "QX_SSC_LED_Red_Online_Q8" := #lfb_blinker_cam.outx_blinker;

	    // FB flash config
	    #lfb_blinker_config(int_periodendauer := T#500ms);

	    //  Deciding which state
	    //  Setup - Calibration State
	    IF "gtyp_Setup".x_Set_Pos_Activ OR "gtyp_Setup".x_Color_Sensor_Calibration
	        OR "gtyp_Setup".x_Counter_Value_Calibration
	        OR "gtyp_Setup".x_Clean_Rack_HBW THEN
	        "QX_SSC_LED_Green_Q5" := #lfb_blinker_config.outx_blinker;
	        "QX_SSC_LED_Yellow_Q6" := #lfb_blinker_config.outx_blinker;
	        "QX_SSC_LED_Red_Q7" := #lfb_blinker_config.outx_blinker;
	        //  Error State
	    ELSIF ("gtyp_Interface_Dashboard".Subscribe.State_HBW.i_code = 4)
	        OR ("gtyp_Interface_Dashboard".Subscribe.State_MPO.i_code = 4)
	        OR ("gtyp_Interface_Dashboard".Subscribe.State_SLD.i_code = 4)
	        OR ("gtyp_Interface_Dashboard".Subscribe.State_VGR.i_code = 4) THEN
	        "QX_SSC_LED_Green_Q5" := FALSE;
	        "QX_SSC_LED_Yellow_Q6" := FALSE;
	        "QX_SSC_LED_Red_Q7" := TRUE;
	        //  Proccessing State
	    ELSIF ("gtyp_Interface_Dashboard".Subscribe.State_HBW.i_code = 2)
	        OR ("gtyp_Interface_Dashboard".Subscribe.State_MPO.i_code = 2)
	        OR ("gtyp_Interface_Dashboard".Subscribe.State_SLD.i_code = 2)
	        OR ("gtyp_Interface_Dashboard".Subscribe.State_VGR.i_code = 2) THEN
	        "QX_SSC_LED_Green_Q5" := FALSE;
	        "QX_SSC_LED_Yellow_Q6" := TRUE;
	        "QX_SSC_LED_Red_Q7" := FALSE;
	        //  Idle State
	    ELSIF ("gtyp_Interface_Dashboard".Subscribe.State_HBW.i_code = 1)
	        AND ("gtyp_Interface_Dashboard".Subscribe.State_MPO.i_code = 1)
	        AND ("gtyp_Interface_Dashboard".Subscribe.State_SLD.i_code = 1)
	        AND ("gtyp_Interface_Dashboard".Subscribe.State_VGR.i_code = 1) THEN
	        "QX_SSC_LED_Green_Q5" := TRUE;
	        "QX_SSC_LED_Yellow_Q6" := FALSE;
	        "QX_SSC_LED_Red_Q7" := FALSE;
	        //  nothing State
	    ELSE
	        "QX_SSC_LED_Green_Q5" := FALSE;
	        "QX_SSC_LED_Yellow_Q6" := FALSE;
	        "QX_SSC_LED_Red_Q7" := FALSE;
	    END_IF;


	ELSE
	    #lx_Init := TRUE;
	END_IF;
END_FUNCTION_BLOCK

FUNCTION_BLOCK "PRG_SSC_Axis_Horizontal"
TITLE = Program Axis horizontal SSC
{ S7_Optimized_Access := 'TRUE' }
AUTHOR : 'A.Schaefer'
VERSION : 0.0
   VAR
      lx_Init { ExternalAccessible := 'False'; ExternalVisible := 'False'; ExternalWritable := 'False'} : Bool;
      lfb_Horizontal_Axis { ExternalAccessible := 'False'; ExternalVisible := 'False'; ExternalWritable := 'False'; S7_SetPoint := 'False'} : "FB_Axis";
   END_VAR


BEGIN
	IF #lx_Init THEN

	    // FB Axis horizontal
	    #lfb_Horizontal_Axis(ini_Axis := 4,
	                         indi_Increment := "gtyp_SSC".Horizontal_Axis.di_Increment,
	                         inx_Ref_Switch := "IX_SSC_RefSwitchHorizontalAxis_I2",
	                         inx_Referencing := "gtyp_SSC".Horizontal_Axis.x_Reference,
	                         inx_Start_Positioning := "gtyp_SSC".Horizontal_Axis.x_Start_Positioning,
	                         indi_Target_Position := "gtyp_SSC".Horizontal_Axis.di_Target_Position,
	                         ini_PWM := "gtyp_SSC".Horizontal_Axis.i_PWM,
	                         inouttyp_Config := "gtyp_SSC".Horizontal_Axis.Config,
	                         inouttyp_Setup := "gtyp_SetupAxis");

	    "QX_SSC_M2_HorizontalAxisCounterclockwise_Q4" := #lfb_Horizontal_Axis.outx_Motor_Neg;
	    "QX_SSC_M2_HorizontalAxisClockwise_Q3" := #lfb_Horizontal_Axis.outx_Motor_Pos;
	    "QW_SSC_PWM_Horizontal_M2" := #lfb_Horizontal_Axis.outi_Motor_PWM;
	    "gtyp_SSC".Horizontal_Axis.di_Actual_Position := #lfb_Horizontal_Axis.outdi_Actual_Position;
	    "gtyp_SSC".Horizontal_Axis.x_Referenced := #lfb_Horizontal_Axis.outx_Referenced;
	    "gtyp_SSC".Horizontal_Axis.x_Position_Reached := #lfb_Horizontal_Axis.outx_Position_Reached;
	ELSE
	    #lx_Init := TRUE;
	END_IF;
END_FUNCTION_BLOCK

FUNCTION_BLOCK "PRG_SSC_Axis_Vertical"
TITLE = Program Axis vertical SSC
{ S7_Optimized_Access := 'TRUE' }
AUTHOR : 'A.Schaefer'
VERSION : 0.0
   VAR
      lx_Init { ExternalAccessible := 'False'; ExternalVisible := 'False'; ExternalWritable := 'False'} : Bool;
      lfb_Vertical_Axis { ExternalAccessible := 'False'; ExternalVisible := 'False'; ExternalWritable := 'False'; S7_SetPoint := 'False'} : "FB_Axis";
   END_VAR


BEGIN
	IF #lx_Init THEN

	    // FB Axis vertical
	    #lfb_Vertical_Axis(ini_Axis := 5,
	                       indi_Increment := "gtyp_SSC".Vertical_Axis.di_Increment,
	                       inx_Ref_Switch := "IX_SSC_RefSwitchVerticalAxis_I1",
	                       inx_Referencing := "gtyp_SSC".Vertical_Axis.x_Reference,
	                       inx_Start_Positioning := "gtyp_SSC".Vertical_Axis.x_Start_Positioning,
	                       indi_Target_Position := "gtyp_SSC".Vertical_Axis.di_Target_Position,
	                       ini_PWM := "gtyp_SSC".Vertical_Axis.i_PWM,
	                       inouttyp_Config := "gtyp_SSC".Vertical_Axis.Config,
	                       inouttyp_Setup := "gtyp_SetupAxis");

	    "QX_SSC_M1_VerticalAxisUp_Q1" := #lfb_Vertical_Axis.outx_Motor_Pos;
	    "QX_SSC_M1_VerticalAxisDown_Q2" := #lfb_Vertical_Axis.outx_Motor_Neg;
	    "QW_SSC_PWM_Vertical_M1" := #lfb_Vertical_Axis.outi_Motor_PWM;
	    "gtyp_SSC".Vertical_Axis.di_Actual_Position := #lfb_Vertical_Axis.outdi_Actual_Position;
	    "gtyp_SSC".Vertical_Axis.x_Referenced := #lfb_Vertical_Axis.outx_Referenced;
	    "gtyp_SSC".Vertical_Axis.x_Position_Reached := #lfb_Vertical_Axis.outx_Position_Reached;
	ELSE
	    #lx_Init := TRUE;
	END_IF;
END_FUNCTION_BLOCK

FUNCTION_BLOCK "PRG_SSC_Calibration_Color"
TITLE = Program Calibration Color Sensor SSC
{ S7_Optimized_Access := 'TRUE' }
AUTHOR : 'A.Schaefer'
VERSION : 0.0
   VAR
      lx_Init { ExternalAccessible := 'False'; ExternalVisible := 'False'; ExternalWritable := 'False'} : Bool;
      lx_Start_TON_Wait { ExternalAccessible := 'False'; ExternalVisible := 'False'; ExternalWritable := 'False'} : Bool;
      lx_Start_Positioning_m { ExternalAccessible := 'False'; ExternalVisible := 'False'; ExternalWritable := 'False'} : Bool;
      lt_TON_Wait { ExternalAccessible := 'False'; ExternalVisible := 'False'; ExternalWritable := 'False'} : Time;
      li_StepCase { ExternalAccessible := 'False'; ExternalVisible := 'False'; ExternalWritable := 'False'} : Int;
      ldi_Pos_Horizontal { ExternalAccessible := 'False'; ExternalVisible := 'False'; ExternalWritable := 'False'} : DInt;
      ldi_Pos_Vertical { ExternalAccessible := 'False'; ExternalVisible := 'False'; ExternalWritable := 'False'} : DInt;
      lfb_R_Trig_Deaktivate {InstructionName := 'R_TRIG'; LibVersion := '1.0'; ExternalAccessible := 'False'; ExternalVisible := 'False'; ExternalWritable := 'False'; S7_SetPoint := 'False'} : R_TRIG;
      lfb_TON_Wait {InstructionName := 'TON_TIME'; LibVersion := '1.0'; ExternalAccessible := 'False'; ExternalVisible := 'False'; ExternalWritable := 'False'; S7_SetPoint := 'False'} : TON_TIME;
   END_VAR


BEGIN
	IF #lx_Init THEN

	    // FB TON Wait
	    #lfb_TON_Wait(IN := #lx_Start_TON_Wait,
	                  PT := #lt_TON_Wait);

	    #lfb_R_Trig_Deaktivate(CLK := NOT "gtyp_Setup".x_Color_Sensor_Calibration
	                           OR NOT ("gtyp_Setup".i_Color_Sensor_Selection = 1));
	    // Deaktivate step 0
	    IF #lfb_R_Trig_Deaktivate.Q THEN
	        "gtyp_Setup".x_Calculate_Value_Color := FALSE;
	        "gtyp_Setup".x_Set_Calib_Value_Color_Blue := FALSE;
	        "gtyp_Setup".x_Set_Calib_Value_Color_Red := FALSE;
	        "gtyp_Setup".x_Set_Calib_Value_Color_White := FALSE;
	        "gtyp_Setup".w_Calib_ColorValue_Blue := 0;
	        "gtyp_Setup".w_Calib_ColorValue_Red := 0;
	        "gtyp_Setup".w_Calib_ColorValue_White := 0;
	        "gtyp_Setup".w_Threshold_Red_Blue := 0;
	        "gtyp_Setup".w_Threshold_White_Red := 0;
	        #li_StepCase := 0;
	    END_IF;

	    // step chain HBW
	    CASE #li_StepCase OF

	        0:  // init
	            #lx_Start_TON_Wait := FALSE;
	            #li_StepCase := 10;

	        10:  // Set Calibration activ?
	            IF "gtyp_Setup".x_Color_Sensor_Calibration
	                AND ("gtyp_Setup".i_Color_Sensor_Selection = 1) THEN
	                "gtyp_Setup".x_Calculate_Value_Color := FALSE;
	                "gtyp_Setup".x_Set_Calib_Value_Color_Blue := FALSE;
	                "gtyp_Setup".x_Set_Calib_Value_Color_Red := FALSE;
	                "gtyp_Setup".x_Set_Calib_Value_Color_White := FALSE;
	                "gtyp_Setup".w_Calib_ColorValue_Blue := 0;
	                "gtyp_Setup".w_Calib_ColorValue_Red := 0;
	                "gtyp_Setup".w_Calib_ColorValue_White := 0;
	                "gtyp_Setup".w_Threshold_Red_Blue := 0;
	                "gtyp_Setup".w_Threshold_White_Red := 0;
	                #li_StepCase := 20;
	            END_IF;

	        20: // wait for set Values or Calculate

	            // Start new Positioning
	            IF "gtyp_Setup".x_Set_Calib_Value_Color_Blue THEN
	                "gtyp_Setup".w_Calib_ColorValue_Blue := "IW_SSC_ColorSensor_A1";
	                "gtyp_Setup".x_Set_Calib_Value_Color_Blue := FALSE;
	            ELSIF "gtyp_Setup".x_Set_Calib_Value_Color_Red THEN
	                "gtyp_Setup".w_Calib_ColorValue_Red := "IW_SSC_ColorSensor_A1";
	                "gtyp_Setup".x_Set_Calib_Value_Color_Red := FALSE;
	            ELSIF "gtyp_Setup".x_Set_Calib_Value_Color_White THEN
	                "gtyp_Setup".w_Calib_ColorValue_White := "IW_SSC_ColorSensor_A1";
	                "gtyp_Setup".x_Set_Calib_Value_Color_White := FALSE;
	            END_IF;

	            "gtyp_Setup".w_Threshold_White_Red := "gtyp_Setup".w_Calib_ColorValue_White + (("gtyp_Setup".w_Calib_ColorValue_Red - "gtyp_Setup".w_Calib_ColorValue_White) / 2);
	            "gtyp_Setup".w_Threshold_Red_Blue := "gtyp_Setup".w_Calib_ColorValue_Red + (("gtyp_Setup".w_Calib_ColorValue_Blue - "gtyp_Setup".w_Calib_ColorValue_Red) / 2);

	            IF "gtyp_Setup".x_Calculate_Value_Color THEN
	                "gtyp_SSC".w_Threshold_White_Red := "gtyp_Setup".w_Threshold_White_Red;
	                "gtyp_SSC".w_Threshold_Red_Blue := "gtyp_Setup".w_Threshold_Red_Blue;
	                "gtyp_Setup".x_Calculate_Value_Color := FALSE;
	            END_IF;

	            // Statement section ELSE
	        ELSE
	            ;
	    END_CASE;

	    IF ("gtyp_Setup".i_Color_Sensor_Selection = 1) THEN
	        // Reload Pos Value
	        "gtyp_Setup".w_Actual_ColorValue := "IW_SSC_ColorSensor_A1";
	    END_IF;
	ELSE
	    #lx_Init := TRUE;
	END_IF;
END_FUNCTION_BLOCK

FUNCTION_BLOCK "PRG_SSC_Set_Park_Position"
TITLE = Program Set Positioning SSC
{ S7_Optimized_Access := 'TRUE' }
AUTHOR : 'A.Schaefer'
VERSION : 0.0
   VAR
      lx_Init { ExternalAccessible := 'False'; ExternalVisible := 'False'; ExternalWritable := 'False'} : Bool;
      lx_Start_TON_Wait { ExternalAccessible := 'False'; ExternalVisible := 'False'; ExternalWritable := 'False'} : Bool;
      lt_TON_Wait { ExternalAccessible := 'False'; ExternalVisible := 'False'; ExternalWritable := 'False'} : Time;
      li_StepCase { ExternalAccessible := 'False'; ExternalVisible := 'False'; ExternalWritable := 'False'} : Int;
      lfb_TON_Wait {InstructionName := 'TON_TIME'; LibVersion := '1.0'; ExternalAccessible := 'False'; ExternalVisible := 'False'; ExternalWritable := 'False'; S7_SetPoint := 'False'} : TON_TIME;
      lfb_R_Trig_Start_Park_Pos {InstructionName := 'R_TRIG'; LibVersion := '1.0'; ExternalAccessible := 'False'; ExternalVisible := 'False'; ExternalWritable := 'False'; S7_SetPoint := 'False'} : R_TRIG;
   END_VAR


BEGIN
	IF #lx_Init THEN

	    // FB TON Wait
	    #lfb_TON_Wait(IN := #lx_Start_TON_Wait,
	                  PT := #lt_TON_Wait);

	    #lfb_R_Trig_Start_Park_Pos(CLK := "gtyp_Setup".x_Park_Position
	                               OR "IX_Set_Park_Position");

	    // Set Start Park Position
	    IF #lfb_R_Trig_Start_Park_Pos.Q THEN
	        "gtyp_SSC".x_Start_Park_Position := TRUE;
	        #li_StepCase := 0;
	    END_IF;

	    // not Start Park Pos Step 0
	    IF NOT "gtyp_SSC".x_Start_Park_Position THEN
	        #li_StepCase := 0;
	    END_IF;

	    // step chain HBW
	    CASE #li_StepCase OF

	        0:  // init
	            #lx_Start_TON_Wait := FALSE;
	            #li_StepCase := 10;

	        10:  // Set Positioning activ?
	            IF "gtyp_SSC".x_Start_Park_Position AND NOT "gtyp_SSC".x_Park_Position_Reached THEN
	                "gtyp_SSC".Horizontal_Axis.x_Start_Positioning := FALSE;
	                "gtyp_SSC".Vertical_Axis.x_Start_Positioning := FALSE;
	                "gtyp_SSC".Horizontal_Axis.x_Reference := FALSE;
	                "gtyp_SSC".Vertical_Axis.x_Reference := FALSE;
	                #li_StepCase := 20;
	            END_IF;

	        20: // homing vertical axis
	            "gtyp_SSC".Vertical_Axis.x_Reference := TRUE;

	            IF NOT "gtyp_SSC".Vertical_Axis.x_Referenced THEN
	                #li_StepCase := 30;
	            END_IF;

	        30: // homed vertical axis
	            IF "gtyp_SSC".Vertical_Axis.x_Referenced THEN
	                "gtyp_SSC".Vertical_Axis.x_Reference := FALSE;
	                #li_StepCase := 40;
	            END_IF;

	        40: // homing horizontal axis
	            "gtyp_SSC".Horizontal_Axis.x_Reference := TRUE;

	            IF NOT "gtyp_SSC".Horizontal_Axis.x_Referenced THEN
	                #li_StepCase := 50;
	            END_IF;

	        50: // homed horizontal axis
	            IF "gtyp_SSC".Horizontal_Axis.x_Referenced THEN
	                "gtyp_SSC".Horizontal_Axis.x_Reference := FALSE;
	                #li_StepCase := 60;
	            END_IF;

	        60: // Position horizontal Axis
	            "gtyp_SSC".Horizontal_Axis.di_Target_Position := "gtyp_SSC".di_Pos_Park_Horizontal;
	            "gtyp_SSC".Horizontal_Axis.x_Start_Positioning := TRUE;

	            IF ("gtyp_SSC".Horizontal_Axis.di_Actual_Position <= ("gtyp_SSC".di_Pos_Park_Horizontal + "gtyp_SSC".Horizontal_Axis.Config.di_Pos_Window))
	                AND ("gtyp_SSC".Horizontal_Axis.di_Actual_Position >= ("gtyp_SSC".di_Pos_Park_Horizontal - "gtyp_SSC".Horizontal_Axis.Config.di_Pos_Window))
	                AND "gtyp_SSC".Horizontal_Axis.x_Position_Reached THEN
	                "gtyp_SSC".Horizontal_Axis.x_Start_Positioning := FALSE;
	                #li_StepCase := 70;
	            END_IF;

	        70: // Position vertical Axis
	            "gtyp_SSC".Vertical_Axis.di_Target_Position := "gtyp_SSC".di_Pos_Park_Vertical;
	            "gtyp_SSC".Vertical_Axis.x_Start_Positioning := TRUE;

	            IF ("gtyp_SSC".Vertical_Axis.di_Actual_Position <= ("gtyp_SSC".di_Pos_Park_Vertical + "gtyp_SSC".Vertical_Axis.Config.di_Pos_Window))
	                AND ("gtyp_SSC".Vertical_Axis.di_Actual_Position >= ("gtyp_SSC".di_Pos_Park_Vertical - "gtyp_SSC".Vertical_Axis.Config.di_Pos_Window))
	                AND "gtyp_SSC".Vertical_Axis.x_Position_Reached THEN
	                "gtyp_SSC".Vertical_Axis.x_Start_Positioning := FALSE;
	                #li_StepCase := 80;
	            END_IF;

	        80: // Deciding which doing
	            "gtyp_SSC".x_Park_Position_Reached := TRUE;


	            // Statement section ELSE
	        ELSE
	            ;
	    END_CASE;

	ELSE
	    #lx_Init := TRUE;
	END_IF;
END_FUNCTION_BLOCK

FUNCTION_BLOCK "PRG_SSC_Set_Positioning"
TITLE = Program Set Positioning SSC
{ S7_Optimized_Access := 'TRUE' }
AUTHOR : 'A.Schaefer'
VERSION : 0.0
   VAR
      lx_Init { ExternalAccessible := 'False'; ExternalVisible := 'False'; ExternalWritable := 'False'} : Bool;
      lx_Start_TON_Wait { ExternalAccessible := 'False'; ExternalVisible := 'False'; ExternalWritable := 'False'} : Bool;
      lx_Start_Positioning_m { ExternalAccessible := 'False'; ExternalVisible := 'False'; ExternalWritable := 'False'} : Bool;
      lt_TON_Wait { ExternalAccessible := 'False'; ExternalVisible := 'False'; ExternalWritable := 'False'} : Time;
      li_StepCase { ExternalAccessible := 'False'; ExternalVisible := 'False'; ExternalWritable := 'False'} : Int;
      ldi_Pos_Horizontal { ExternalAccessible := 'False'; ExternalVisible := 'False'; ExternalWritable := 'False'} : DInt;
      ldi_Pos_Vertical { ExternalAccessible := 'False'; ExternalVisible := 'False'; ExternalWritable := 'False'} : DInt;
      lfb_R_Trig_Deaktivate {InstructionName := 'R_TRIG'; LibVersion := '1.0'; ExternalAccessible := 'False'; ExternalVisible := 'False'; ExternalWritable := 'False'; S7_SetPoint := 'False'} : R_TRIG;
      lfb_TON_Wait {InstructionName := 'TON_TIME'; LibVersion := '1.0'; ExternalAccessible := 'False'; ExternalVisible := 'False'; ExternalWritable := 'False'; S7_SetPoint := 'False'} : TON_TIME;
   END_VAR


BEGIN
	IF #lx_Init THEN

	    // FB TON Wait
	    #lfb_TON_Wait(IN := #lx_Start_TON_Wait,
	                  PT := #lt_TON_Wait);

	    #lfb_R_Trig_Deaktivate(CLK := NOT "gtyp_Setup".x_Set_Pos_Activ
	                           OR NOT (("gtyp_Setup".i_Pos_Selection > 0)
	                           AND ("gtyp_Setup".i_Pos_Selection < 21)));
	    // Deaktivate step 10
	    IF #lfb_R_Trig_Deaktivate.Q THEN
	        "gtyp_SSC".Horizontal_Axis.x_Start_Positioning := FALSE;
	        "gtyp_SSC".Vertical_Axis.x_Start_Positioning := FALSE;
	        "gtyp_SSC".Horizontal_Axis.x_Reference := FALSE;
	        "gtyp_SSC".Vertical_Axis.x_Reference := FALSE;
	        "gtyp_Setup".x_Start_Positioning := FALSE;
	        "gtyp_Setup".x_Final_Positioning := FALSE;
	        "gtyp_Setup".x_Home_Positioning := FALSE;
	        "gtyp_Setup".x_Start_Offset := FALSE;
	        #lx_Start_Positioning_m := FALSE;
	        IF (#li_StepCase > 10) THEN
	            #li_StepCase := 70;
	        END_IF;
	    END_IF;

	    // Set Positioning activ?
	    IF "gtyp_Setup".x_Set_Pos_Activ
	        AND (("gtyp_Setup".i_Pos_Selection > 0)
	        AND ("gtyp_Setup".i_Pos_Selection < 21))
	        AND ((#li_StepCase = 40)
	        OR (#li_StepCase = 60)) THEN

	        // Deciding which Position
	        // Position - Centre
	        IF "gtyp_Setup".i_Pos_Selection = 1 THEN
	            #ldi_Pos_Horizontal := "gtyp_SSC".di_Pos_Centre_Horizontal;
	            #ldi_Pos_Vertical := "gtyp_SSC".di_Pos_Centre_Vertical;
	            // Position - HBW
	        ELSIF "gtyp_Setup".i_Pos_Selection = 2 THEN
	            #ldi_Pos_Horizontal := "gtyp_SSC".di_Pos_HBW_Horizontal;
	            #ldi_Pos_Vertical := "gtyp_SSC".di_Pos_HBW_Vertical;
	        END_IF;
	    END_IF;

	    // Set Positioning activ?
	    IF NOT "gtyp_Setup".x_Set_Pos_Activ THEN
	        "gtyp_Setup".i_Pos_Selection := 0;
	    END_IF;

	    // step chain HBW
	    CASE #li_StepCase OF

	        0:  // init
	            #lx_Start_TON_Wait := FALSE;
	            #li_StepCase := 10;

	        10:  // Set Positioning activ?
	            IF "gtyp_Setup".x_Set_Pos_Activ
	                AND (("gtyp_Setup".i_Pos_Selection > 0)
	                AND ("gtyp_Setup".i_Pos_Selection < 21)) THEN
	                "gtyp_SSC".Horizontal_Axis.x_Start_Positioning := FALSE;
	                "gtyp_SSC".Vertical_Axis.x_Start_Positioning := FALSE;
	                "gtyp_SSC".Horizontal_Axis.x_Reference := FALSE;
	                "gtyp_SSC".Vertical_Axis.x_Reference := FALSE;
	                "gtyp_Setup".x_Start_Positioning := FALSE;
	                "gtyp_Setup".x_Final_Positioning := FALSE;
	                "gtyp_Setup".x_Home_Positioning := FALSE;
	                "gtyp_Setup".x_Start_Offset := FALSE;
	                #li_StepCase := 20;
	            END_IF;

	        20: //homing vertical/horizontal axis

	            "gtyp_SSC".Horizontal_Axis.x_Reference := TRUE;
	            "gtyp_SSC".Vertical_Axis.x_Reference := TRUE;

	            IF NOT "gtyp_SSC".Horizontal_Axis.x_Referenced AND NOT "gtyp_SSC".Vertical_Axis.x_Referenced THEN
	                #li_StepCase := 30;
	            END_IF;

	        30: // homed vertical/horizontal axis
	            IF "gtyp_SSC".Horizontal_Axis.x_Referenced THEN
	                "gtyp_SSC".Horizontal_Axis.x_Reference := FALSE;
	            END_IF;
	            IF "gtyp_SSC".Vertical_Axis.x_Referenced THEN
	                "gtyp_SSC".Vertical_Axis.x_Reference := FALSE;
	            END_IF;

	            IF "gtyp_SSC".Horizontal_Axis.x_Referenced AND "gtyp_SSC".Vertical_Axis.x_Referenced THEN
	                "gtyp_SSC".Horizontal_Axis.x_Reference := FALSE;
	                "gtyp_SSC".Vertical_Axis.x_Reference := FALSE;
	                #li_StepCase := 40;
	            END_IF;

	        40:  // Start Positioning Step next
	            IF "gtyp_Setup".x_Start_Positioning OR #lx_Start_Positioning_m THEN
	                #lx_Start_Positioning_m := FALSE;
	                #li_StepCase := 50;
	            END_IF;

	        50: // Position vertical/horizontal HBW
	            "gtyp_SSC".Horizontal_Axis.di_Target_Position := #ldi_Pos_Horizontal;
	            "gtyp_SSC".Horizontal_Axis.x_Start_Positioning := TRUE;
	            "gtyp_SSC".Vertical_Axis.di_Target_Position := #ldi_Pos_Vertical;
	            "gtyp_SSC".Vertical_Axis.x_Start_Positioning := TRUE;

	            IF ("gtyp_SSC".Horizontal_Axis.di_Actual_Position <= (#ldi_Pos_Horizontal + "gtyp_SSC".Horizontal_Axis.Config.di_Pos_Window))
	                AND ("gtyp_SSC".Horizontal_Axis.di_Actual_Position >= (#ldi_Pos_Horizontal - "gtyp_SSC".Horizontal_Axis.Config.di_Pos_Window))
	                AND "gtyp_SSC".Horizontal_Axis.x_Position_Reached THEN
	                "gtyp_SSC".Horizontal_Axis.x_Start_Positioning := FALSE;
	            END_IF;

	            IF ("gtyp_SSC".Vertical_Axis.di_Actual_Position <= (#ldi_Pos_Vertical + "gtyp_SSC".Vertical_Axis.Config.di_Pos_Window))
	                AND ("gtyp_SSC".Vertical_Axis.di_Actual_Position >= (#ldi_Pos_Vertical - "gtyp_SSC".Vertical_Axis.Config.di_Pos_Window))
	                AND "gtyp_SSC".Vertical_Axis.x_Position_Reached THEN
	                "gtyp_SSC".Vertical_Axis.x_Start_Positioning := FALSE;
	            END_IF;

	            IF ("gtyp_SSC".Horizontal_Axis.di_Actual_Position <= (#ldi_Pos_Horizontal + "gtyp_SSC".Horizontal_Axis.Config.di_Pos_Window))
	                AND ("gtyp_SSC".Horizontal_Axis.di_Actual_Position >= (#ldi_Pos_Horizontal - "gtyp_SSC".Horizontal_Axis.Config.di_Pos_Window))
	                AND "gtyp_SSC".Horizontal_Axis.x_Position_Reached
	                AND ("gtyp_SSC".Vertical_Axis.di_Actual_Position <= (#ldi_Pos_Vertical + "gtyp_SSC".Vertical_Axis.Config.di_Pos_Window))
	                AND ("gtyp_SSC".Vertical_Axis.di_Actual_Position >= (#ldi_Pos_Vertical - "gtyp_SSC".Vertical_Axis.Config.di_Pos_Window))
	                AND "gtyp_SSC".Vertical_Axis.x_Position_Reached THEN
	                "gtyp_SSC".Horizontal_Axis.x_Start_Positioning := FALSE;
	                "gtyp_SSC".Vertical_Axis.x_Start_Positioning := FALSE;
	                "gtyp_Setup".x_Start_Positioning := FALSE;
	                #li_StepCase := 60;
	            END_IF;

	        60: // Deciding which doing

	            // Start new Positioning
	            IF "gtyp_Setup".x_Start_Positioning OR "gtyp_Setup".x_Home_Positioning THEN
	                #lx_Start_Positioning_m := TRUE;
	                #li_StepCase := 10;
	            ELSIF #lfb_R_Trig_Deaktivate.Q THEN
	                "gtyp_Setup".x_Home_Positioning := FALSE;
	                #li_StepCase := 70;
	            END_IF;

	        70: //homing vertical/horizontal axis

	            "gtyp_SSC".Horizontal_Axis.x_Reference := TRUE;
	            "gtyp_SSC".Vertical_Axis.x_Reference := TRUE;

	            IF NOT "gtyp_SSC".Horizontal_Axis.x_Referenced AND NOT "gtyp_SSC".Vertical_Axis.x_Referenced THEN
	                #li_StepCase := 80;
	            END_IF;

	        80: // homed vertical/horizontal axis
	            IF "gtyp_SSC".Horizontal_Axis.x_Referenced THEN
	                "gtyp_SSC".Horizontal_Axis.x_Reference := FALSE;
	            END_IF;
	            IF "gtyp_SSC".Vertical_Axis.x_Referenced THEN
	                "gtyp_SSC".Vertical_Axis.x_Reference := FALSE;
	            END_IF;

	            IF "gtyp_SSC".Horizontal_Axis.x_Referenced AND "gtyp_SSC".Vertical_Axis.x_Referenced THEN
	                "gtyp_SSC".Horizontal_Axis.x_Reference := FALSE;
	                "gtyp_SSC".Vertical_Axis.x_Reference := FALSE;
	                #li_StepCase := 0;
	            END_IF;

	            // Statement section ELSE
	        ELSE
	            ;
	    END_CASE;

	    IF (("gtyp_Setup".i_Pos_Selection > 0)
	        AND ("gtyp_Setup".i_Pos_Selection < 21)) THEN
	        // Reload Pos Value
	        "gtyp_Setup".di_Pos_Horizontal := #ldi_Pos_Horizontal;
	        "gtyp_Setup".di_Pos_Vertical := #ldi_Pos_Vertical;
	        "gtyp_Setup".di_Pos_Rotate := 0;
	    END_IF;
	ELSE
	    #lx_Init := TRUE;
	END_IF;
END_FUNCTION_BLOCK

FUNCTION_BLOCK "PRG_SSC_Ablauf"
TITLE = Program Ablauf SSC
{ S7_Optimized_Access := 'TRUE' }
AUTHOR : 'A.Schaefer'
VERSION : 0.0
   VAR
      lx_Init { ExternalAccessible := 'False'; ExternalVisible := 'False'; ExternalWritable := 'False'} : Bool;
      lx_FirstCentre { ExternalAccessible := 'False'; ExternalVisible := 'False'; ExternalWritable := 'False'} : Bool;
      lx_Start { ExternalAccessible := 'False'; ExternalVisible := 'False'; ExternalWritable := 'False'} : Bool;
      lx_Start_TON_State { ExternalAccessible := 'False'; ExternalVisible := 'False'; ExternalWritable := 'False'} : Bool;
      lt_TON_Wait { ExternalAccessible := 'False'; ExternalVisible := 'False'; ExternalWritable := 'False'} : Time;
      li_StepCase { ExternalAccessible := 'False'; ExternalVisible := 'False'; ExternalWritable := 'False'} : Int;
      ldi_TargetPosition_Horizontal { ExternalAccessible := 'False'; ExternalVisible := 'False'; ExternalWritable := 'False'} : DInt;
      ldi_TargetPosition_Vertical { ExternalAccessible := 'False'; ExternalVisible := 'False'; ExternalWritable := 'False'} : DInt;
      lldt_ts_old { ExternalAccessible := 'False'; ExternalVisible := 'False'; ExternalWritable := 'False'} : LDT;
      ldt_write { ExternalAccessible := 'False'; ExternalVisible := 'False'; ExternalWritable := 'False'} : Date_And_Time;
      li_Return_write { ExternalAccessible := 'False'; ExternalVisible := 'False'; ExternalWritable := 'False'} : Int;
      ldt_MQTT { ExternalAccessible := 'False'; ExternalVisible := 'False'; ExternalWritable := 'False'} : Date_And_Time;
      li_Return_LDT { ExternalAccessible := 'False'; ExternalVisible := 'False'; ExternalWritable := 'False'} : Int;
      lx_Start_TON_Wait { ExternalAccessible := 'False'; ExternalVisible := 'False'; ExternalWritable := 'False'} : Bool;
      ldi_StepHorizontal { ExternalAccessible := 'False'; ExternalVisible := 'False'; ExternalWritable := 'False'} : DInt;
      ldi_StepVertical { ExternalAccessible := 'False'; ExternalVisible := 'False'; ExternalWritable := 'False'} : DInt;
      lfb_TON_Wait {InstructionName := 'TON_TIME'; LibVersion := '1.0'; ExternalAccessible := 'False'; ExternalVisible := 'False'; ExternalWritable := 'False'; S7_SetPoint := 'False'} : TON_TIME;
      lfb_TON_State {InstructionName := 'TON_TIME'; LibVersion := '1.0'; ExternalAccessible := 'False'; ExternalVisible := 'False'; ExternalWritable := 'False'; S7_SetPoint := 'False'} : TON_TIME;
      lfb_F_TRIG_Set_Pos {InstructionName := 'F_TRIG'; LibVersion := '1.0'; ExternalAccessible := 'False'; ExternalVisible := 'False'; ExternalWritable := 'False'; S7_SetPoint := 'False'} : F_TRIG;
   END_VAR


BEGIN
	IF #lx_Init THEN

	    // Restart after set Positioning
	    IF "gtyp_Setup".x_Set_Pos_Activ OR "gtyp_SSC".x_Start_Park_Position THEN
	        #li_StepCase := 0;
	    END_IF;

	    // falling edge Set Pos
	    #lfb_F_TRIG_Set_Pos(CLK := "gtyp_Setup".x_Set_Pos_Activ);

	    IF #lfb_F_TRIG_Set_Pos.Q THEN
	        #lx_FirstCentre := TRUE;
	    END_IF;

	    #lfb_TON_Wait(IN := #lx_Start_TON_Wait,
	                  PT := #lt_TON_Wait);

	    // wait time state
	    #lfb_TON_State(IN := NOT #lx_Start_TON_State,
	                   PT := T#2s);

	    // state of the ssc cyclically transmitted to the cloud
	    IF #lfb_TON_State.Q AND NOT #lx_Start_TON_State THEN
	        #lx_Start_TON_State := TRUE;
	        #li_Return_LDT := RD_SYS_T(#ldt_MQTT);
	        "gtyp_Interface_Dashboard".Subscribe.PosPanTiltUnit.ldt_ts := DT_TO_LDT(#ldt_MQTT);
	    END_IF;

	    // restart wait time state
	    IF NOT #lfb_TON_State.Q AND #lx_Start_TON_State THEN
	        #lx_Start_TON_State := FALSE;
	    END_IF;

	    CASE #li_StepCase OF

	        0:  // Init
	            #lx_Start_TON_State := FALSE;
	            "gtyp_SSC".Horizontal_Axis.x_Start_Positioning := FALSE;
	            "gtyp_SSC".Vertical_Axis.x_Start_Positioning := FALSE;

	            IF NOT "gtyp_Setup".x_Set_Pos_Activ AND NOT "gtyp_SSC".x_Start_Park_Position THEN
	                #li_StepCase := 10;
	            END_IF;

	        10: // Deciding which route to take

	            IF ("gtyp_Interface_Dashboard".Publish.PosPanTiltUnit.ldt_ts > #lldt_ts_old) OR #lx_FirstCentre THEN

	                #lldt_ts_old := "gtyp_Interface_Dashboard".Publish.PosPanTiltUnit.ldt_ts;

	                // convert the degrees to position
	                #ldi_StepHorizontal := REAL_TO_DINT("FC_Scale_linear"(inr_Y1 := DINT_TO_REAL("gtyp_SSC".Horizontal_Axis.Config.di_Neg_Soft_Switch),
	                                                                                                          inr_Y2 := DINT_TO_REAL("gtyp_SSC".Horizontal_Axis.Config.di_Pos_Soft_Switch),
	                                                                                                          inr_X1 := 0.0,
	                                                                                                          inr_X2 := 180.0,
	                                                                                                          inr_X := DINT_TO_REAL("gtyp_Interface_Dashboard".Publish.PosPanTiltUnit.i_degree)));
	                #ldi_StepVertical := REAL_TO_DINT("FC_Scale_linear"(inr_Y1 := DINT_TO_REAL("gtyp_SSC".Vertical_Axis.Config.di_Neg_Soft_Switch),
	                                                                                                      inr_Y2 := DINT_TO_REAL("gtyp_SSC".Vertical_Axis.Config.di_Pos_Soft_Switch),
	                                                                                                      inr_X1 := 0.0,
	                                                                                                      inr_X2 := 180.0,
	                                                                                                      inr_X := DINT_TO_REAL("gtyp_Interface_Dashboard".Publish.PosPanTiltUnit.i_degree)));
	                // Procedure - relmove_left
	                IF ("gtyp_Interface_Dashboard".Publish.PosPanTiltUnit.s_cmd = 'relmove_left')
	                    AND (("gtyp_SSC".Horizontal_Axis.di_Actual_Position - #ldi_StepHorizontal) > "gtyp_SSC".Horizontal_Axis.Config.di_Neg_Soft_Switch + 15)
	                    AND NOT "IX_SSC_RefSwitchHorizontalAxis_I2" THEN
	                    #ldi_TargetPosition_Horizontal := "gtyp_SSC".Horizontal_Axis.di_Actual_Position - #ldi_StepHorizontal;
	                    "gtyp_SSC".Horizontal_Axis.di_Target_Position := #ldi_TargetPosition_Horizontal;
	                    "gtyp_SSC".Horizontal_Axis.x_Start_Positioning := TRUE;
	                    #li_StepCase := 70;
	                    // Procedure - relmove_right
	                ELSIF ("gtyp_Interface_Dashboard".Publish.PosPanTiltUnit.s_cmd = 'relmove_right')
	                    AND (("gtyp_SSC".Horizontal_Axis.di_Actual_Position + #ldi_StepHorizontal) < "gtyp_SSC".Horizontal_Axis.Config.di_Pos_Soft_Switch - 15) THEN
	                    #ldi_TargetPosition_Horizontal := "gtyp_SSC".Horizontal_Axis.di_Actual_Position + #ldi_StepHorizontal;
	                    "gtyp_SSC".Horizontal_Axis.di_Target_Position := #ldi_TargetPosition_Horizontal;
	                    "gtyp_SSC".Horizontal_Axis.x_Start_Positioning := TRUE;
	                    #li_StepCase := 70;
	                    // Procedure - relmove_up
	                ELSIF ("gtyp_Interface_Dashboard".Publish.PosPanTiltUnit.s_cmd = 'relmove_up')
	                    AND (("gtyp_SSC".Vertical_Axis.di_Actual_Position + #ldi_StepHorizontal) < "gtyp_SSC".Vertical_Axis.Config.di_Pos_Soft_Switch - 15) THEN
	                    #ldi_TargetPosition_Vertical := "gtyp_SSC".Vertical_Axis.di_Actual_Position + #ldi_StepVertical;
	                    "gtyp_SSC".Vertical_Axis.di_Target_Position := #ldi_TargetPosition_Vertical;
	                    "gtyp_SSC".Vertical_Axis.x_Start_Positioning := TRUE;
	                    #li_StepCase := 80;
	                    // Procedure - relmove_down
	                ELSIF ("gtyp_Interface_Dashboard".Publish.PosPanTiltUnit.s_cmd = 'relmove_down')
	                    AND (("gtyp_SSC".Vertical_Axis.di_Actual_Position - #ldi_StepVertical) > "gtyp_SSC".Vertical_Axis.Config.di_Neg_Soft_Switch + 15)
	                    AND NOT "IX_SSC_RefSwitchVerticalAxis_I1" THEN
	                    #ldi_TargetPosition_Vertical := "gtyp_SSC".Vertical_Axis.di_Actual_Position - #ldi_StepVertical;
	                    "gtyp_SSC".Vertical_Axis.di_Target_Position := #ldi_TargetPosition_Vertical;
	                    "gtyp_SSC".Vertical_Axis.x_Start_Positioning := TRUE;
	                    #li_StepCase := 80;
	                    // Procedure - first
	                ELSIF #lx_FirstCentre THEN
	                    #li_StepCase := 20;
	                    // Procedure - home
	                ELSIF ("gtyp_Interface_Dashboard".Publish.PosPanTiltUnit.s_cmd = 'home') THEN
	                    #li_StepCase := 60;
	                    // Procedure - start_pan
	                ELSIF ("gtyp_Interface_Dashboard".Publish.PosPanTiltUnit.s_cmd = 'start_pan')
	                    AND ("gtyp_SSC".Horizontal_Axis.di_Actual_Position > "gtyp_SSC".Horizontal_Axis.Config.di_Neg_Soft_Switch + 15)
	                    AND NOT "IX_SSC_RefSwitchHorizontalAxis_I2" THEN
	                    #ldi_TargetPosition_Horizontal := "gtyp_SSC".Horizontal_Axis.Config.di_Neg_Soft_Switch + 15;
	                    "gtyp_SSC".Horizontal_Axis.di_Target_Position := #ldi_TargetPosition_Horizontal;
	                    "gtyp_SSC".Horizontal_Axis.x_Start_Positioning := TRUE;
	                    #li_StepCase := 70;
	                    // Procedure - end_pan
	                ELSIF ("gtyp_Interface_Dashboard".Publish.PosPanTiltUnit.s_cmd = 'end_pan')
	                    AND ("gtyp_SSC".Horizontal_Axis.di_Actual_Position < "gtyp_SSC".Horizontal_Axis.Config.di_Pos_Soft_Switch - 15) THEN
	                    #ldi_TargetPosition_Horizontal := "gtyp_SSC".Horizontal_Axis.Config.di_Pos_Soft_Switch - 15;
	                    "gtyp_SSC".Horizontal_Axis.di_Target_Position := #ldi_TargetPosition_Horizontal;
	                    "gtyp_SSC".Horizontal_Axis.x_Start_Positioning := TRUE;
	                    #li_StepCase := 70;
	                    // Procedure - start_tilt
	                ELSIF ("gtyp_Interface_Dashboard".Publish.PosPanTiltUnit.s_cmd = 'start_tilt')
	                    AND ("gtyp_SSC".Vertical_Axis.di_Actual_Position > "gtyp_SSC".Vertical_Axis.Config.di_Neg_Soft_Switch + 15)
	                    AND NOT "IX_SSC_RefSwitchVerticalAxis_I1" THEN
	                    #ldi_TargetPosition_Vertical := "gtyp_SSC".Vertical_Axis.Config.di_Neg_Soft_Switch + 15;
	                    "gtyp_SSC".Vertical_Axis.di_Target_Position := #ldi_TargetPosition_Vertical;
	                    "gtyp_SSC".Vertical_Axis.x_Start_Positioning := TRUE;
	                    #li_StepCase := 80;
	                    // Procedure - end_tilt
	                ELSIF ("gtyp_Interface_Dashboard".Publish.PosPanTiltUnit.s_cmd = 'end_tilt')
	                    AND ("gtyp_SSC".Vertical_Axis.di_Actual_Position < "gtyp_SSC".Vertical_Axis.Config.di_Pos_Soft_Switch - 15) THEN
	                    #ldi_TargetPosition_Vertical := "gtyp_SSC".Vertical_Axis.Config.di_Pos_Soft_Switch - 15;
	                    "gtyp_SSC".Vertical_Axis.di_Target_Position := #ldi_TargetPosition_Vertical;
	                    "gtyp_SSC".Vertical_Axis.x_Start_Positioning := TRUE;
	                    #li_StepCase := 80;
	                END_IF;
	            END_IF;

	        20: // homing vertical/horizontal axis
	            "gtyp_SSC".Horizontal_Axis.x_Reference := TRUE;
	            "gtyp_SSC".Vertical_Axis.x_Reference := TRUE;

	            IF NOT "gtyp_SSC".Horizontal_Axis.x_Referenced AND NOT "gtyp_SSC".Vertical_Axis.x_Referenced THEN
	                #li_StepCase := 30;
	            END_IF;

	        30: // homed vertical/horizontal axis
	            IF "gtyp_SSC".Horizontal_Axis.x_Referenced THEN
	                "gtyp_SSC".Horizontal_Axis.x_Reference := FALSE;
	            END_IF;
	            IF "gtyp_SSC".Vertical_Axis.x_Referenced THEN
	                "gtyp_SSC".Vertical_Axis.x_Reference := FALSE;
	            END_IF;

	            IF "gtyp_SSC".Horizontal_Axis.x_Referenced AND "gtyp_SSC".Vertical_Axis.x_Referenced THEN
	                "gtyp_SSC".Horizontal_Axis.x_Reference := FALSE;
	                "gtyp_SSC".Vertical_Axis.x_Reference := FALSE;
	                #lx_Start_TON_Wait := TRUE;
	                #li_StepCase := 40;
	            END_IF;

	        40: // wait sequence
	            IF #lfb_TON_Wait.Q THEN
	                #lx_Start_TON_Wait := FALSE;
	                #li_StepCase := 50;
	            END_IF;

	        50: // Position horizontal/vertical axis and reached
	            "gtyp_SSC".Horizontal_Axis.di_Target_Position := "gtyp_SSC".di_Pos_HBW_Horizontal;
	            "gtyp_SSC".Horizontal_Axis.x_Start_Positioning := TRUE;
	            "gtyp_SSC".Vertical_Axis.di_Target_Position := "gtyp_SSC".di_Pos_HBW_Vertical;
	            "gtyp_SSC".Vertical_Axis.x_Start_Positioning := TRUE;

	            IF ("gtyp_SSC".Horizontal_Axis.di_Actual_Position <= ("gtyp_SSC".di_Pos_HBW_Horizontal + "gtyp_SSC".Horizontal_Axis.Config.di_Pos_Window))
	                AND ("gtyp_SSC".Horizontal_Axis.di_Actual_Position >= ("gtyp_SSC".di_Pos_HBW_Horizontal - "gtyp_SSC".Horizontal_Axis.Config.di_Pos_Window))
	                AND "gtyp_SSC".Horizontal_Axis.x_Position_Reached THEN
	                "gtyp_SSC".Horizontal_Axis.x_Start_Positioning := FALSE;
	            END_IF;

	            IF ("gtyp_SSC".Vertical_Axis.di_Actual_Position <= ("gtyp_SSC".di_Pos_HBW_Vertical + "gtyp_SSC".Vertical_Axis.Config.di_Pos_Window))
	                AND ("gtyp_SSC".Vertical_Axis.di_Actual_Position >= ("gtyp_SSC".di_Pos_HBW_Vertical - "gtyp_SSC".Vertical_Axis.Config.di_Pos_Window))
	                AND "gtyp_SSC".Vertical_Axis.x_Position_Reached THEN
	                "gtyp_SSC".Vertical_Axis.x_Start_Positioning := FALSE;
	            END_IF;

	            IF ("gtyp_SSC".Horizontal_Axis.di_Actual_Position <= ("gtyp_SSC".di_Pos_HBW_Horizontal + "gtyp_SSC".Horizontal_Axis.Config.di_Pos_Window))
	                AND ("gtyp_SSC".Horizontal_Axis.di_Actual_Position >= ("gtyp_SSC".di_Pos_HBW_Horizontal - "gtyp_SSC".Horizontal_Axis.Config.di_Pos_Window))
	                AND "gtyp_SSC".Horizontal_Axis.x_Position_Reached
	                AND ("gtyp_SSC".Vertical_Axis.di_Actual_Position <= ("gtyp_SSC".di_Pos_HBW_Vertical + "gtyp_SSC".Vertical_Axis.Config.di_Pos_Window))
	                AND ("gtyp_SSC".Vertical_Axis.di_Actual_Position >= ("gtyp_SSC".di_Pos_HBW_Vertical - "gtyp_SSC".Vertical_Axis.Config.di_Pos_Window))
	                AND "gtyp_SSC".Vertical_Axis.x_Position_Reached THEN
	                "gtyp_SSC".Horizontal_Axis.x_Start_Positioning := FALSE;
	                "gtyp_SSC".Vertical_Axis.x_Start_Positioning := FALSE;
	                #lx_FirstCentre := FALSE;
	                #li_StepCase := 90;
	            END_IF;

	        60: // Position Centre horizontal/vertical axis and reached
	            "gtyp_SSC".Horizontal_Axis.di_Target_Position := "gtyp_SSC".di_Pos_Centre_Horizontal;
	            "gtyp_SSC".Horizontal_Axis.x_Start_Positioning := TRUE;
	            "gtyp_SSC".Vertical_Axis.di_Target_Position := "gtyp_SSC".di_Pos_Centre_Vertical;
	            "gtyp_SSC".Vertical_Axis.x_Start_Positioning := TRUE;

	            IF ("gtyp_SSC".Horizontal_Axis.di_Actual_Position <= ("gtyp_SSC".di_Pos_Centre_Horizontal + "gtyp_SSC".Horizontal_Axis.Config.di_Pos_Window))
	                AND ("gtyp_SSC".Horizontal_Axis.di_Actual_Position >= ("gtyp_SSC".di_Pos_Centre_Horizontal - "gtyp_SSC".Horizontal_Axis.Config.di_Pos_Window))
	                AND "gtyp_SSC".Horizontal_Axis.x_Position_Reached THEN
	                "gtyp_SSC".Horizontal_Axis.x_Start_Positioning := FALSE;
	            END_IF;

	            IF ("gtyp_SSC".Vertical_Axis.di_Actual_Position <= ("gtyp_SSC".di_Pos_Centre_Vertical + "gtyp_SSC".Vertical_Axis.Config.di_Pos_Window))
	                AND ("gtyp_SSC".Vertical_Axis.di_Actual_Position >= ("gtyp_SSC".di_Pos_Centre_Vertical - "gtyp_SSC".Vertical_Axis.Config.di_Pos_Window))
	                AND "gtyp_SSC".Vertical_Axis.x_Position_Reached THEN
	                "gtyp_SSC".Vertical_Axis.x_Start_Positioning := FALSE;
	            END_IF;

	            IF ("gtyp_SSC".Horizontal_Axis.di_Actual_Position <= ("gtyp_SSC".di_Pos_Centre_Horizontal + "gtyp_SSC".Horizontal_Axis.Config.di_Pos_Window))
	                AND ("gtyp_SSC".Horizontal_Axis.di_Actual_Position >= ("gtyp_SSC".di_Pos_Centre_Horizontal - "gtyp_SSC".Horizontal_Axis.Config.di_Pos_Window))
	                AND "gtyp_SSC".Horizontal_Axis.x_Position_Reached
	                AND ("gtyp_SSC".Vertical_Axis.di_Actual_Position <= ("gtyp_SSC".di_Pos_Centre_Vertical + "gtyp_SSC".Vertical_Axis.Config.di_Pos_Window))
	                AND ("gtyp_SSC".Vertical_Axis.di_Actual_Position >= ("gtyp_SSC".di_Pos_Centre_Vertical - "gtyp_SSC".Vertical_Axis.Config.di_Pos_Window))
	                AND "gtyp_SSC".Vertical_Axis.x_Position_Reached THEN
	                "gtyp_SSC".Horizontal_Axis.x_Start_Positioning := FALSE;
	                "gtyp_SSC".Vertical_Axis.x_Start_Positioning := FALSE;
	                #lx_FirstCentre := FALSE;
	                #li_StepCase := 90;
	            END_IF;

	        70: // Position horizontal axis reached
	            IF ("gtyp_SSC".Horizontal_Axis.di_Actual_Position <= (#ldi_TargetPosition_Horizontal + "gtyp_SSC".Horizontal_Axis.Config.di_Pos_Window))
	                AND ("gtyp_SSC".Horizontal_Axis.di_Actual_Position >= (#ldi_TargetPosition_Horizontal - "gtyp_SSC".Horizontal_Axis.Config.di_Pos_Window))
	                AND "gtyp_SSC".Horizontal_Axis.x_Position_Reached THEN
	                "gtyp_SSC".Horizontal_Axis.x_Start_Positioning := FALSE;
	                #li_StepCase := 90;
	            END_IF;

	        80: // Position vertical axis reached
	            IF ("gtyp_SSC".Vertical_Axis.di_Actual_Position <= (#ldi_TargetPosition_Vertical + "gtyp_SSC".Vertical_Axis.Config.di_Pos_Window))
	                AND ("gtyp_SSC".Vertical_Axis.di_Actual_Position >= (#ldi_TargetPosition_Vertical - "gtyp_SSC".Vertical_Axis.Config.di_Pos_Window))
	                AND "gtyp_SSC".Vertical_Axis.x_Position_Reached THEN
	                "gtyp_SSC".Vertical_Axis.x_Start_Positioning := FALSE;
	                #li_StepCase := 90;
	            END_IF;

	        90: // convert the position to degrees
	            "gtyp_Interface_Dashboard".Subscribe.PosPanTiltUnit.r_pan := "FC_Scale_linear"(inr_Y1 := -1.0,
	                                                                                           inr_Y2 := 1.0,
	                                                                                           inr_X1 := DINT_TO_REAL("gtyp_SSC".Horizontal_Axis.Config.di_Neg_Soft_Switch),
	                                                                                           inr_X2 := DINT_TO_REAL("gtyp_SSC".Horizontal_Axis.Config.di_Pos_Soft_Switch),
	                                                                                           inr_X := "gtyp_SSC".Horizontal_Axis.di_Actual_Position);
	            "gtyp_Interface_Dashboard".Subscribe.PosPanTiltUnit.r_tilt := "FC_Scale_linear"(inr_Y1 := -1.0,
	                                                                                            inr_Y2 := 1.0,
	                                                                                            inr_X1 := DINT_TO_REAL("gtyp_SSC".Vertical_Axis.Config.di_Neg_Soft_Switch),
	                                                                                            inr_X2 := DINT_TO_REAL("gtyp_SSC".Vertical_Axis.Config.di_Pos_Soft_Switch),
	                                                                                            inr_X := "gtyp_SSC".Vertical_Axis.di_Actual_Position);

	            #li_Return_write := RD_SYS_T(#ldt_write);
	            "gtyp_Interface_Dashboard".Subscribe.PosPanTiltUnit.ldt_ts := DT_TO_LDT(#ldt_write);
	            #lx_Start_TON_Wait := TRUE;
	            #li_StepCase := 100;

	        100:// wait sequence
	            IF #lfb_TON_Wait.Q THEN
	                #lx_Start_TON_Wait := FALSE;
	                #li_StepCase := 0;
	            END_IF;
	            // Statement section ELSE
	        ELSE
	            ;
	    END_CASE;

	ELSE
	    #lx_Init := TRUE;
	    #lx_FirstCentre := TRUE;

	    "gtyp_SSC".x_Start_Park_Position := FALSE;
	    "gtyp_SSC".x_Park_Position_Reached := FALSE;
	    "gtyp_SSC".x_Error := FALSE;
	END_IF;
END_FUNCTION_BLOCK

FUNCTION_BLOCK "PRG_VGR_Set_Positioning"
TITLE = Program Set Positioning VGR
{ S7_Optimized_Access := 'TRUE' }
AUTHOR : 'A.Schaefer'
VERSION : 0.0
   VAR
      lx_Init { ExternalAccessible := 'False'; ExternalVisible := 'False'; ExternalWritable := 'False'} : Bool;
      lx_Start_TON_Wait { ExternalAccessible := 'False'; ExternalVisible := 'False'; ExternalWritable := 'False'} : Bool;
      lx_Start_Positioning_m { ExternalAccessible := 'False'; ExternalVisible := 'False'; ExternalWritable := 'False'} : Bool;
      lx_Start_FinalPositioning_m { ExternalAccessible := 'False'; ExternalVisible := 'False'; ExternalWritable := 'False'} : Bool;
      lx_Start_TON_State { ExternalAccessible := 'False'; ExternalVisible := 'False'; ExternalWritable := 'False'} : Bool;
      lt_TON_Wait { ExternalAccessible := 'False'; ExternalVisible := 'False'; ExternalWritable := 'False'} : Time;
      ldt_MQTT { ExternalAccessible := 'False'; ExternalVisible := 'False'; ExternalWritable := 'False'} : Date_And_Time;
      li_Return_LDT { ExternalAccessible := 'False'; ExternalVisible := 'False'; ExternalWritable := 'False'} : Int;
      li_Lights { ExternalAccessible := 'False'; ExternalVisible := 'False'; ExternalWritable := 'False'} : Int;
      li_Lights_old { ExternalAccessible := 'False'; ExternalVisible := 'False'; ExternalWritable := 'False'} : Int;
      lx_State_activ { ExternalAccessible := 'False'; ExternalVisible := 'False'; ExternalWritable := 'False'} : Bool;
      li_StepCase { ExternalAccessible := 'False'; ExternalVisible := 'False'; ExternalWritable := 'False'} : Int;
      li_Counter { ExternalAccessible := 'False'; ExternalVisible := 'False'; ExternalWritable := 'False'} : Int;
      ldi_Pos_SLD_X { ExternalAccessible := 'False'; ExternalVisible := 'False'; ExternalWritable := 'False'} : DInt;
      ldi_Pos_SLD_Y { ExternalAccessible := 'False'; ExternalVisible := 'False'; ExternalWritable := 'False'} : DInt;
      ldi_Pos_SLD_Z { ExternalAccessible := 'False'; ExternalVisible := 'False'; ExternalWritable := 'False'} : DInt;
      ldi_Pos_Horizontal { ExternalAccessible := 'False'; ExternalVisible := 'False'; ExternalWritable := 'False'} : DInt;
      ldi_Pos_Vertical { ExternalAccessible := 'False'; ExternalVisible := 'False'; ExternalWritable := 'False'} : DInt;
      ldi_Pos_Rotate { ExternalAccessible := 'False'; ExternalVisible := 'False'; ExternalWritable := 'False'} : DInt;
      ldi_Offset_Vertical { ExternalAccessible := 'False'; ExternalVisible := 'False'; ExternalWritable := 'False'} : DInt;
      ls_Color { ExternalAccessible := 'False'; ExternalVisible := 'False'; ExternalWritable := 'False'} : String;
      ls_Target { ExternalAccessible := 'False'; ExternalVisible := 'False'; ExternalWritable := 'False'} : String;
      lfb_TON_Wait {InstructionName := 'TON_TIME'; LibVersion := '1.0'; ExternalAccessible := 'False'; ExternalVisible := 'False'; ExternalWritable := 'False'; S7_SetPoint := 'False'} : TON_TIME;
      lfb_TON_State {InstructionName := 'TON_TIME'; LibVersion := '1.0'; ExternalAccessible := 'False'; ExternalVisible := 'False'; ExternalWritable := 'False'; S7_SetPoint := 'False'} : TON_TIME;
      lfb_R_Trig_Deaktivate {InstructionName := 'R_TRIG'; LibVersion := '1.0'; ExternalAccessible := 'False'; ExternalVisible := 'False'; ExternalWritable := 'False'; S7_SetPoint := 'False'} : R_TRIG;
      lfb_R_Trig_NiO {InstructionName := 'R_TRIG'; LibVersion := '1.0'; ExternalAccessible := 'False'; ExternalVisible := 'False'; ExternalWritable := 'False'; S7_SetPoint := 'False'} : R_TRIG;
   END_VAR


BEGIN
	IF #lx_Init THEN

	    // FB TON Wait
	    #lfb_TON_Wait(IN := #lx_Start_TON_Wait,
	                  PT := #lt_TON_Wait);

	    #lfb_R_Trig_Deaktivate(CLK := NOT "gtyp_Setup".x_Set_Pos_Activ
	                           OR NOT (("gtyp_Setup".i_Pos_Selection > 40)
	                           AND ("gtyp_Setup".i_Pos_Selection < 61)));
	    // Deaktivate step 150
	    IF #lfb_R_Trig_Deaktivate.Q THEN
	        "gtyp_VGR".horizontal_Axis.x_Start_Positioning := FALSE;
	        "gtyp_VGR".vertical_Axis.x_Start_Positioning := FALSE;
	        "gtyp_VGR".rotate_Axis.x_Start_Positioning := FALSE;
	        "gtyp_VGR".horizontal_Axis.x_Reference := FALSE;
	        "gtyp_VGR".vertical_Axis.x_Reference := FALSE;
	        "gtyp_VGR".rotate_Axis.x_Reference := FALSE;
	        "gtyp_Setup".x_Start_Positioning := FALSE;
	        "gtyp_Setup".x_Final_Positioning := FALSE;
	        "gtyp_Setup".x_Home_Positioning := FALSE;
	        "gtyp_Setup".x_Start_Offset := FALSE;
	        IF (#li_StepCase > 10) THEN
	            #li_StepCase := 150;
	        END_IF;
	    END_IF;

	    // Set Positioning activ?
	    IF "gtyp_Setup".x_Set_Pos_Activ
	        AND (("gtyp_Setup".i_Pos_Selection > 40)
	        AND ("gtyp_Setup".i_Pos_Selection < 61))
	        AND ((#li_StepCase = 80)
	        OR (#li_StepCase = 120)
	        OR (#li_StepCase = 140)) THEN

	        // Deciding which Position
	        // Position - Color
	        IF "gtyp_Setup".i_Pos_Selection = 41 THEN
	            #ldi_Pos_Horizontal := "gtyp_VGR".di_Pos_Color_horizontal;
	            #ldi_Pos_Vertical := "gtyp_VGR".di_Pos_Color_vertical;
	            #ldi_Pos_Rotate := "gtyp_VGR".di_Pos_Color_rotate;
	            #ldi_Offset_Vertical := "gtyp_VGR".di_Offset_Pos_DSI_NFC_vertical;
	            // Position - DSI Collect
	        ELSIF "gtyp_Setup".i_Pos_Selection = 42 THEN
	            #ldi_Pos_Horizontal := "gtyp_VGR".di_Pos_DSI_horizontal;
	            #ldi_Pos_Vertical := "gtyp_VGR".di_Pos_DSI_Collect_vertical;
	            #ldi_Pos_Rotate := "gtyp_VGR".di_Pos_DSI_rotate;
	            #ldi_Offset_Vertical := "gtyp_VGR".di_Offset_Pos_DSI_NFC_vertical;
	            // Position - DSI Discard
	        ELSIF "gtyp_Setup".i_Pos_Selection = 43 THEN
	            #ldi_Pos_Horizontal := "gtyp_VGR".di_Pos_DSI_horizontal;
	            #ldi_Pos_Vertical := "gtyp_VGR".di_Pos_DSI_Discard_vertical;
	            #ldi_Pos_Rotate := "gtyp_VGR".di_Pos_DSI_rotate;
	            #ldi_Offset_Vertical := "gtyp_VGR".di_Offset_Pos_DSI_NFC_vertical;
	            // Position - DSO Collect
	        ELSIF "gtyp_Setup".i_Pos_Selection = 44 THEN
	            #ldi_Pos_Horizontal := "gtyp_VGR".di_Pos_DSO_horizontal;
	            #ldi_Pos_Vertical := "gtyp_VGR".di_Pos_DSO_Collect_vertical;
	            #ldi_Pos_Rotate := "gtyp_VGR".di_Pos_DSO_rotate;
	            #ldi_Offset_Vertical := "gtyp_VGR".di_Offset_Pos_DSO_vertical;
	            // Position - DSO Discard
	        ELSIF "gtyp_Setup".i_Pos_Selection = 45 THEN
	            #ldi_Pos_Horizontal := "gtyp_VGR".di_Pos_DSO_horizontal;
	            #ldi_Pos_Vertical := "gtyp_VGR".di_Pos_DSO_Discard_vertical;
	            #ldi_Pos_Rotate := "gtyp_VGR".di_Pos_DSO_rotate;
	            #ldi_Offset_Vertical := "gtyp_VGR".di_Offset_Pos_DSO_vertical;
	            // Position - HBW Collect
	        ELSIF "gtyp_Setup".i_Pos_Selection = 46 THEN
	            #ldi_Pos_Horizontal := "gtyp_VGR".di_Pos_HBW_horizontal;
	            #ldi_Pos_Vertical := "gtyp_VGR".di_Pos_HBW_Collect_vertical;
	            #ldi_Pos_Rotate := "gtyp_VGR".di_Pos_HBW_rotate;
	            #ldi_Offset_Vertical := "gtyp_VGR".di_Offset_Pos_HBW_vertical;
	            // Position - HBW Discard
	        ELSIF "gtyp_Setup".i_Pos_Selection = 47 THEN
	            #ldi_Pos_Horizontal := "gtyp_VGR".di_Pos_HBW_horizontal;
	            #ldi_Pos_Vertical := "gtyp_VGR".di_Pos_HBW_Discard_vertical;
	            #ldi_Pos_Rotate := "gtyp_VGR".di_Pos_HBW_rotate;
	            #ldi_Offset_Vertical := "gtyp_VGR".di_Offset_Pos_HBW_vertical;
	            // Position - MPO
	        ELSIF "gtyp_Setup".i_Pos_Selection = 48 THEN
	            #ldi_Pos_Horizontal := "gtyp_VGR".di_Pos_MPO_horizontal;
	            #ldi_Pos_Vertical := "gtyp_VGR".di_Pos_MPO_vertical;
	            #ldi_Pos_Rotate := "gtyp_VGR".di_Pos_MPO_rotate;
	            #ldi_Offset_Vertical := "gtyp_VGR".di_Offset_Pos_MPO_vertical;
	            // Position - NFC
	        ELSIF "gtyp_Setup".i_Pos_Selection = 49 THEN
	            #ldi_Pos_Horizontal := "gtyp_VGR".di_Pos_NFC_horizontal;
	            #ldi_Pos_Vertical := "gtyp_VGR".di_Pos_NFC_vertical;
	            #ldi_Pos_Rotate := "gtyp_VGR".di_Pos_NFC_rotate;
	            #ldi_Offset_Vertical := "gtyp_VGR".di_Offset_Pos_DSI_NFC_vertical;
	            // Position - NiO
	        ELSIF "gtyp_Setup".i_Pos_Selection = 50 THEN
	            #ldi_Pos_Horizontal := "gtyp_VGR".di_Pos_NiO_horizontal;
	            #ldi_Pos_Vertical := "gtyp_VGR".di_Pos_NiO_vertical;
	            #ldi_Pos_Rotate := "gtyp_VGR".di_Pos_NiO_rotate;
	            #ldi_Offset_Vertical := 500;
	            // Position - SLD Blue
	        ELSIF "gtyp_Setup".i_Pos_Selection = 51 THEN
	            #ldi_Pos_Horizontal := "gtyp_VGR".di_Pos_SLD_Blue_horizontal;
	            #ldi_Pos_Vertical := "gtyp_VGR".di_Pos_SLD_Blue_vertical;
	            #ldi_Pos_Rotate := "gtyp_VGR".di_Pos_SLD_Blue_rotate;
	            #ldi_Offset_Vertical := 500;
	            // Position - SLD Red
	        ELSIF "gtyp_Setup".i_Pos_Selection = 52 THEN
	            #ldi_Pos_Horizontal := "gtyp_VGR".di_Pos_SLD_Red_horizontal;
	            #ldi_Pos_Vertical := "gtyp_VGR".di_Pos_SLD_Red_vertical;
	            #ldi_Pos_Rotate := "gtyp_VGR".di_Pos_SLD_Red_rotate;
	            #ldi_Offset_Vertical := 500;
	            // Position - SLD White
	        ELSIF "gtyp_Setup".i_Pos_Selection = 53 THEN
	            #ldi_Pos_Horizontal := "gtyp_VGR".di_Pos_SLD_White_horizontal;
	            #ldi_Pos_Vertical := "gtyp_VGR".di_Pos_SLD_White_vertical;
	            #ldi_Pos_Rotate := "gtyp_VGR".di_Pos_SLD_White_rotate;
	            #ldi_Offset_Vertical := 500;
	        END_IF;
	    END_IF;

	    // Set Positioning activ?
	    IF NOT "gtyp_Setup".x_Set_Pos_Activ THEN
	        "gtyp_Setup".i_Pos_Selection := 0;
	    END_IF;

	    // step chain HBW
	    CASE #li_StepCase OF

	        0:  // init
	            #lx_Start_TON_Wait := FALSE;
	            #li_StepCase := 10;

	        10:  // Set Positioning activ?
	            IF "gtyp_Setup".x_Set_Pos_Activ
	                AND (("gtyp_Setup".i_Pos_Selection > 40)
	                AND ("gtyp_Setup".i_Pos_Selection < 61)) THEN

	                "gtyp_VGR".horizontal_Axis.x_Start_Positioning := FALSE;
	                "gtyp_VGR".vertical_Axis.x_Start_Positioning := FALSE;
	                "gtyp_VGR".rotate_Axis.x_Start_Positioning := FALSE;
	                "gtyp_VGR".horizontal_Axis.x_Reference := FALSE;
	                "gtyp_VGR".vertical_Axis.x_Reference := FALSE;
	                "gtyp_VGR".rotate_Axis.x_Reference := FALSE;
	                "gtyp_Setup".x_Start_Positioning := FALSE;
	                "gtyp_Setup".x_Final_Positioning := FALSE;
	                "gtyp_Setup".x_Home_Positioning := FALSE;
	                "gtyp_Setup".x_Start_Offset := FALSE;
	                "gtyp_VGR".vertical_Axis.i_PWM := 800;
	                #li_StepCase := 20;
	            END_IF;

	        20: // homing vertical axis
	            "gtyp_VGR".vertical_Axis.x_Reference := TRUE;

	            IF NOT "gtyp_VGR".vertical_Axis.x_Referenced THEN
	                #li_StepCase := 30;
	            END_IF;

	        30: // homed vertical axis
	            IF "gtyp_VGR".vertical_Axis.x_Referenced THEN
	                "gtyp_VGR".vertical_Axis.x_Reference := FALSE;
	                #li_StepCase := 40;
	            END_IF;

	        40: // homing horizontal axis
	            "gtyp_VGR".horizontal_Axis.x_Reference := TRUE;

	            IF NOT "gtyp_VGR".horizontal_Axis.x_Referenced THEN
	                #li_StepCase := 50;
	            END_IF;

	        50: // homed horizontal axis
	            IF "gtyp_VGR".horizontal_Axis.x_Referenced THEN
	                "gtyp_VGR".horizontal_Axis.x_Reference := FALSE;
	                #li_StepCase := 60;
	            END_IF;

	        60: // homing rotate axis
	            "gtyp_VGR".rotate_Axis.x_Reference := TRUE;

	            IF NOT "gtyp_VGR".rotate_Axis.x_Referenced THEN
	                #li_StepCase := 70;
	            END_IF;

